KUKA KRL program: MyProgram_189().src

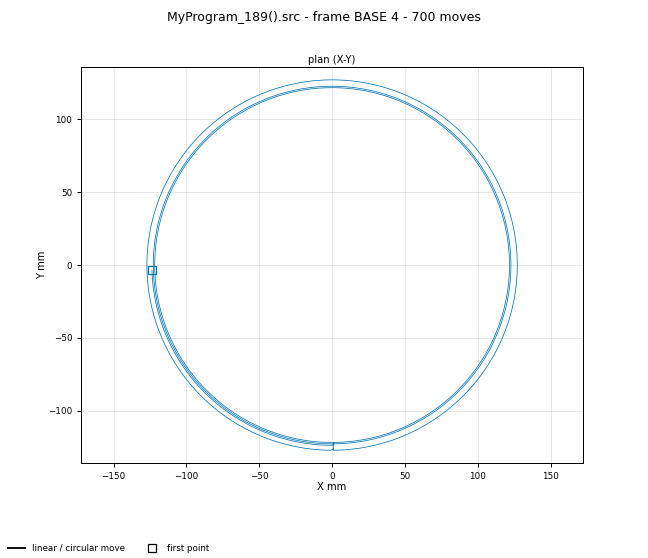
[picture p0: tool path of MyProgram_189().src in frame BASE 4, 700 of 700 moves have a stored position in this frame; points joined in program order, loops and branches not executed]
&ACCESS RVP
&REL 1
&PARAM TEMPLATE = C:\KRC\Roboter\Template\vorgabe
&PARAM EDITMASK = *
DEF MyProgram_189()
; ---- Setting reference (Base) ----
$BASE = BASE_DATA[4]

; --------------------------
; ---- Setting tool (TCP) ----
$TOOL = TOOL_DATA[3]
; --------------------------

$VEL.CP = VEL_APROX_PRINT
Startdeposition()
$VEL.CP = VEL_PRINT
LIN {X -123.6871,Y -3.6269,Z 137,A 178.2903,B 24.9532,C -1.5798,E1 24.8398,E2 627.9376} C_DIS
LIN {X -123.3118,Y -10.2868,Z 137,A -177.6765,B 24.9513,C -1.6119,E1 24.8407,E2 623.8034} C_DIS
LIN {X -122.6788,Y -16.1715,Z 137,A -175.7764,B 24.9541,C -1.5654,E1 24.8413,E2 622.0029} C_DIS
LIN {X -121.5631,Y -23.1085,Z 137,A -172.7109,B 24.9552,C -1.5466,E1 24.8427,E2 618.9641} C_DIS
LIN {X -120.6893,Y -27.3078,Z 137,A -170.7718,B 24.9557,C -1.5382,E1 24.8439,E2 617.0335} C_DIS
LIN {X -120.022,Y -30.1061,Z 137,A -169.137,B 24.9551,C -1.5475,E1 24.8449,E2 615.367} C_DIS
LIN {X -119.1579,Y -33.3607,Z 137,A -167.6264,B 24.9555,C -1.5405,E1 24.8461,E2 613.8643} C_DIS
LIN {X -118.1442,Y -36.7947,Z 137,A -165.8598,B 24.9555,C -1.5402,E1 24.8475,E2 612.0882} C_DIS
LIN {X -116.8715,Y -40.6521,Z 137,A -164.0681,B 24.9561,C -1.5305,E1 24.8491,E2 610.3094} C_DIS
LIN {X -115.0667,Y -45.5133,Z 137,A -161.702,B 24.9566,C -1.5218,E1 24.8514,E2 607.9509} C_DIS
LIN {X -113.3795,Y -49.5667,Z 137,A -159.0001,B 24.9552,C -1.5459,E1 24.8545,E2 605.1764} C_DIS
LIN {X -111.5077,Y -53.6436,Z 137,A -157.538,B 24.9572,C -1.5122,E1 24.8562,E2 603.7867} C_DIS
LIN {X -110.1039,Y -56.4691,Z 137,A -155.9162,B 24.957,C -1.5153,E1 24.8582,E2 602.1488} C_DIS
LIN {X -107.9699,Y -60.4525,Z 137,A -153.8399,B 24.9574,C -1.5088,E1 24.861,E2 600.0772} C_DIS
LIN {X -105.7639,Y -64.2339,Z 137,A -151.6138,B 24.9572,C -1.5123,E1 24.8642,E2 597.8311} C_DIS
LIN {X -103.0515,Y -68.5012,Z 137,A -149.4533,B 24.958,C -1.4979,E1 24.8675,E2 595.694} C_DIS
LIN {X -101.0702,Y -71.3917,Z 137,A -147.7939,B 24.9581,C -1.4955,E1 24.8701,E2 594.0324} C_DIS
LIN {X -98.5873,Y -74.7836,Z 137,A -145.5061,B 24.9575,C -1.5062,E1 24.874,E2 591.708} C_DIS
LIN {X -96.2651,Y -77.7495,Z 137,A -144.2835,B 24.9591,C -1.4782,E1 24.8761,E2 590.5464} C_DIS
LIN {X -94.0528,Y -80.4124,Z 137,A -142.028,B 24.9576,C -1.5042,E1 24.8803,E2 588.2186} C_DIS
LIN {X -91.1944,Y -83.6394,Z 137,A -140.5066,B 24.9591,C -1.4779,E1 24.883,E2 586.7531} C_DIS
LIN {X -88.2872,Y -86.7026,Z 137,A -138.5112,B 24.9592,C -1.4754,E1 24.8869,E2 584.7551} C_DIS
LIN {X -84.7954,Y -90.1202,Z 137,A -136.2459,B 24.9595,C -1.4708,E1 24.8915,E2 582.4914} C_DIS
LIN {X -81.9301,Y -92.733,Z 137,A -134.2054,B 24.9591,C -1.4784,E1 24.8958,E2 580.4245} C_DIS
LIN {X -79.4553,Y -94.8621,Z 137,A -132.7772,B 24.9594,C -1.4716,E1 24.8988,E2 579.007} C_DIS
LIN {X -76.1,Y -97.575,Z 137,A -130.9012,B 24.9599,C -1.4623,E1 24.9029,E2 577.1463} C_DIS
LIN {X -71.8228,Y -100.7645,Z 137,A -128.2909,B 24.9599,C -1.4644,E1 24.9088,E2 574.5216} C_DIS
LIN {X -68.6261,Y -102.9681,Z 137,A -126.6407,B 24.9604,C -1.4546,E1 24.9126,E2 572.8893} C_DIS
LIN {X -63.7724,Y -106.043,Z 137,A -124.2535,B 24.9613,C -1.4378,E1 24.9182,E2 570.5346} C_DIS
LIN {X -60.1181,Y -108.1564,Z 137,A -122.1093,B 24.9609,C -1.4438,E1 24.9234,E2 568.3698} C_DIS
LIN {X -56.5383,Y -110.0687,Z 137,A -120.1188,B 24.9609,C -1.4465,E1 24.9283,E2 566.3673} C_DIS
LIN {X -53.3181,Y -111.6632,Z 137,A -118.5447,B 24.9611,C -1.4403,E1 24.9323,E2 564.8039} C_DIS
LIN {X -50.4843,Y -112.9727,Z 137,A -117.1034,B 24.9612,C -1.4385,E1 24.9359,E2 563.3635} C_DIS
LIN {X -47.5297,Y -114.2474,Z 137,A -115.6287,B 24.9614,C -1.4361,E1 24.9397,E2 561.8909} C_DIS
LIN {X -44.917,Y -115.2996,Z 137,A -114.3059,B 24.9614,C -1.4357,E1 24.9432,E2 560.5662} C_DIS
LIN {X -41.6351,Y -116.5254,Z 137,A -112.6718,B 24.9614,C -1.4348,E1 24.9474,E2 558.931} C_DIS
LIN {X -38.2424,Y -117.6836,Z 137,A -110.1543,B 24.9593,C -1.4744,E1 24.9544,E2 556.3149} C_DIS
LIN {X -32.6953,Y -119.344,Z 137,A -107.5652,B 24.9596,C -1.4682,E1 24.9613,E2 553.7364} C_DIS
LIN {X -27.6129,Y -120.6196,Z 137,A -106.2171,B 24.9625,C -1.4153,E1 24.9647,E2 552.5121} C_DIS
LIN {X -24.7432,Y -121.2408,Z 137,A -104.5438,B 24.9617,C -1.4296,E1 24.9693,E2 550.8029} C_DIS
LIN {X -21.8539,Y -121.7948,Z 137,A -103.1642,B 24.9617,C -1.4299,E1 24.9731,E2 549.421} C_DIS
LIN {X -18.5585,Y -122.3409,Z 137,A -101.5093,B 24.9614,C -1.4347,E1 24.9777,E2 547.7533} C_DIS
LIN {X -14.6586,Y -122.8687,Z 137,A -99.7775,B 24.9617,C -1.43,E1 24.9825,E2 546.0315} C_DIS
LIN {X -10.8263,Y -123.2662,Z 137,A -97.9502,B 24.9616,C -1.4319,E1 24.9876,E2 544.1986} C_DIS
LIN {X -7.19,Y -123.5317,Z 137,A -96.2218,B 24.9615,C -1.4339,E1 24.9924,E2 542.4649} C_DIS
LIN {X -3.2774,Y -123.6968,Z 137,A -94.53,B 24.9618,C -1.4282,E1 24.9971,E2 540.7862} C_DIS
LIN {X 0.3681,Y -123.74,Z 137,A -92.7859,B 24.9616,C -1.4313,E1 25.002,E2 539.0349} C_DIS
LIN {X 0.3681,Y -123.74,Z 137,A -92.7859,B 24.9616,C -1.4313,E1 25.002,E2 539.0349} C_DIS
Enddeposition()
LIN {X 0.8758,Y -122.7486,Z 137,A -93.1134,B 24.7966,C -1.3866,E1 24.8338,E2 539.4449} C_DIS
Startdeposition()
$VEL.CP = VEL_PRINT
LIN {X -2.203,Y -122.7353,Z 137,A -94.7816,B 24.7972,C -1.3754,E1 24.829,E2 541.1399} C_DIS
LIN {X -6.2,Y -122.5983,Z 137,A -96.5836,B 24.797,C -1.3783,E1 24.824,E2 542.9354} C_DIS
LIN {X -10.1585,Y -122.3339,Z 137,A -98.4379,B 24.797,C -1.3782,E1 24.8188,E2 544.7908} C_DIS
LIN {X -13.8748,Y -121.97,Z 137,A -100.0956,B 24.7968,C -1.3823,E1 24.8143,E2 546.4395} C_DIS
LIN {X -16.3768,Y -121.6582,Z 137,A -101.2545,B 24.7968,C -1.3834,E1 24.8111,E2 547.5966} C_DIS
LIN {X -19.0663,Y -121.2654,Z 137,A -102.6876,B 24.7972,C -1.3761,E1 24.8071,E2 549.0485} C_DIS
LIN {X -23.0341,Y -120.5743,Z 137,A -104.5963,B 24.7972,C -1.3755,E1 24.8018,E2 550.9607} C_DIS
LIN {X -26.3906,Y -119.8854,Z 137,A -106.3525,B 24.7975,C -1.3689,E1 24.797,E2 552.7346} C_DIS
LIN {X -31.0253,Y -118.7709,Z 137,A -108.4556,B 24.7972,C -1.3758,E1 24.7913,E2 554.8243} C_DIS
LIN {X -36.1084,Y -117.3239,Z 137,A -110.7655,B 24.7967,C -1.3848,E1 24.7852,E2 557.1166} C_DIS
LIN {X -39.4539,Y -116.2436,Z 137,A -112.57,B 24.797,C -1.3786,E1 24.7803,E2 558.9394} C_DIS
LIN {X -43.2692,Y -114.876,Z 137,A -114.3597,B 24.7967,C -1.385,E1 24.7757,E2 560.7174} C_DIS
LIN {X -47.3278,Y -113.264,Z 137,A -116.3718,B 24.7965,C -1.3883,E1 24.7705,E2 562.7262} C_DIS
LIN {X -50.4824,Y -111.8943,Z 137,A -118.082,B 24.7967,C -1.3853,E1 24.7661,E2 564.4477} C_DIS
LIN {X -54.3057,Y -110.0888,Z 137,A -120.0413,B 24.7965,C -1.3883,E1 24.7611,E2 566.4047} C_DIS
LIN {X -58.3909,Y -107.9802,Z 137,A -122.2379,B 24.7965,C -1.3889,E1 24.7557,E2 568.6062} C_DIS
LIN {X -61.4605,Y -106.2625,Z 137,A -123.6618,B 24.7959,C -1.401,E1 24.7523,E2 570.0052} C_DIS
LIN {X -64.4498,Y -104.4767,Z 137,A -125.4217,B 24.796,C -1.3974,E1 24.7481,E2 571.7793} C_DIS
LIN {X -66.9121,Y -102.9168,Z 137,A -126.6891,B 24.7957,C -1.4037,E1 24.7451,E2 573.0356} C_DIS
LIN {X -70.0256,Y -100.8242,Z 137,A -128.5719,B 24.7959,C -1.4007,E1 24.7408,E2 574.932} C_DIS
LIN {X -73.4065,Y -98.3901,Z 137,A -130.4788,B 24.7956,C -1.4058,E1 24.7365,E2 576.8335} C_DIS
LIN {X -76.3345,Y -96.1362,Z 137,A -132.99,B 24.7973,C -1.3741,E1 24.7308,E2 579.43} C_DIS
LIN {X -80.5143,Y -92.664,Z 137,A -134.5604,B 24.7947,C -1.4218,E1 24.7277,E2 580.8922} C_DIS
LIN {X -82.724,Y -90.6969,Z 137,A -136.647,B 24.7963,C -1.3933,E1 24.7232,E2 583.0555} C_DIS
LIN {X -85.7181,Y -87.8727,Z 137,A -138.0889,B 24.7949,C -1.4185,E1 24.7204,E2 584.4431} C_DIS
LIN {X -88.4014,Y -85.1726,Z 137,A -139.9578,B 24.7949,C -1.4183,E1 24.7167,E2 586.3205} C_DIS
LIN {X -92.3318,Y -80.895,Z 137,A -142.3613,B 24.7939,C -1.4381,E1 24.7123,E2 588.6874} C_DIS
LIN {X -95.0176,Y -77.7224,Z 137,A -144.8359,B 24.7949,C -1.4192,E1 24.7078,E2 591.2188} C_DIS
LIN {X -98.2431,Y -73.6039,Z 137,A -147.0598,B 24.794,C -1.4347,E1 24.704,E2 593.4162} C_DIS
LIN {X -100.2392,Y -70.8606,Z 137,A -148.6789,B 24.794,C -1.4372,E1 24.7014,E2 595.0374} C_DIS
LIN {X -102.6767,Y -67.2806,Z 137,A -150.6986,B 24.7936,C -1.4425,E1 24.6983,E2 597.0544} C_DIS
LIN {X -104.7284,Y -64.0399,Z 137,A -152.4277,B 24.7932,C -1.4499,E1 24.6957,E2 598.7747} C_DIS
LIN {X -106.8253,Y -60.4779,Z 137,A -154.4607,B 24.7932,C -1.4507,E1 24.6929,E2 600.8165} C_DIS
LIN {X -108.9144,Y -56.6265,Z 137,A -156.3406,B 24.7925,C -1.4636,E1 24.6904,E2 602.6756} C_DIS
LIN {X -110.111,Y -54.2606,Z 137,A -157.5975,B 24.7923,C -1.4663,E1 24.6889,E2 603.9328} C_DIS
LIN {X -112.469,Y -49.19,Z 137,A -160.1364,B 24.7917,C -1.4768,E1 24.6859,E2 606.4604} C_DIS
LIN {X -114.1297,Y -45.2066,Z 137,A -162.5726,B 24.7924,C -1.4645,E1 24.6833,E2 608.9399} C_DIS
LIN {X -115.6223,Y -41.2351,Z 137,A -164.2347,B 24.7913,C -1.4842,E1 24.6818,E2 610.5642} C_DIS
LIN {X -116.4754,Y -38.7577,Z 137,A -165.5381,B 24.7913,C -1.4844,E1 24.6806,E2 611.8745} C_DIS
LIN {X -117.6988,Y -34.8687,Z 137,A -167.4771,B 24.7911,C -1.4887,E1 24.679,E2 613.8145} C_DIS
LIN {X -118.6317,Y -31.5472,Z 137,A -169.0788,B 24.7908,C -1.4941,E1 24.6778,E2 615.4128} C_DIS
LIN {X -119.3871,Y -28.5564,Z 137,A -170.4849,B 24.7904,C -1.5,E1 24.6769,E2 616.8129} C_DIS
LIN {X -120.248,Y -24.6815,Z 137,A -172.3898,B 24.7902,C -1.5036,E1 24.6758,E2 618.7204} C_DIS
LIN {X -121.2683,Y -19.0474,Z 137,A -174.8254,B 24.7892,C -1.5223,E1 24.6746,E2 621.1257} C_DIS
LIN {X -121.6872,Y -16.1555,Z 137,A -177.037,B 24.791,C -1.4904,E1 24.6737,E2 623.4272} C_DIS
LIN {X -122.1963,Y -11.6968,Z 137,A -178.4788,B 24.789,C -1.525,E1 24.6734,E2 624.7946} C_DIS
LIN {X -122.6145,Y -5.8764,Z 137,A 178.5874,B 24.789,C -1.5248,E1 24.6728,E2 627.7467} C_DIS
LIN {X -122.7397,Y 1.9378,Z 137,A 174.6848,B 24.789,C -1.5259,E1 24.6728,E2 631.6704} C_DIS
LIN {X -122.64,Y 5.3393,Z 137,A 173.499,B 24.7876,C -1.5483,E1 24.6728,E2 632.8097} C_DIS
LIN {X -122.4564,Y 8.564,Z 137,A 171.4913,B 24.7886,C -1.5319,E1 24.6733,E2 634.8689} C_DIS
LIN {X -122.1415,Y 12.268,Z 137,A 170.293,B 24.7869,C -1.5605,E1 24.6736,E2 636.0059} C_DIS
LIN {X -121.5349,Y 17.2629,Z 137,A 168.0484,B 24.7862,C -1.5726,E1 24.6743,E2 638.2348} C_DIS
LIN {X -121.1308,Y 19.9036,Z 137,A 166.5383,B 24.7866,C -1.5654,E1 24.675,E2 639.7714} C_DIS
LIN {X -120.4521,Y 23.672,Z 137,A 164.4795,B 24.787,C -1.5596,E1 24.6761,E2 641.8564} C_DIS
LIN {X -119.5012,Y 28.0833,Z 137,A 162.5098,B 24.7862,C -1.5722,E1 24.6773,E2 643.8075} C_DIS
LIN {X -118.5997,Y 31.6672,Z 137,A 160.9056,B 24.7856,C -1.583,E1 24.6784,E2 645.3953} C_DIS
LIN {X -117.6401,Y 35.0693,Z 137,A 158.6514,B 24.7868,C -1.5625,E1 24.6802,E2 647.7118} C_DIS
LIN {X -116.3206,Y 39.2222,Z 137,A 157.2285,B 24.7849,C -1.5949,E1 24.6814,E2 649.0649} C_DIS
LIN {X -115.2329,Y 42.3153,Z 137,A 155.3591,B 24.7855,C -1.5852,E1 24.6832,E2 650.9683} C_DIS
LIN {X -113.6971,Y 46.2798,Z 137,A 153.5156,B 24.7847,C -1.5974,E1 24.6851,E2 652.7929} C_DIS
LIN {X -112.1953,Y 49.8095,Z 137,A 151.7129,B 24.7844,C -1.6024,E1 24.6871,E2 654.5937} C_DIS
LIN {X -110.2535,Y 53.9717,Z 137,A 149.805,B 24.7834,C -1.6191,E1 24.6894,E2 656.4721} C_DIS
LIN {X -108.7234,Y 56.9901,Z 137,A 148.0972,B 24.7834,C -1.6183,E1 24.6916,E2 658.1909} C_DIS
LIN {X -104.3676,Y 64.6266,Z 137,A 144.018,B 24.7827,C -1.6313,E1 24.6973,E2 662.2604} C_DIS
LIN {X -100.8109,Y 70.0449,Z 137,A 141.0126,B 24.7821,C -1.6407,E1 24.7019,E2 665.2584} C_DIS
LIN {X -99.122,Y 72.4157,Z 137,A 139.4708,B 24.7823,C -1.6365,E1 24.7044,E2 666.8178} C_DIS
LIN {X -96.7658,Y 75.5356,Z 137,A 137.5795,B 24.7823,C -1.6386,E1 24.7077,E2 668.7132} C_DIS
LIN {X -93.9199,Y 79.0455,Z 137,A 135.5122,B 24.7817,C -1.646,E1 24.7113,E2 670.7723} C_DIS
LIN {X -91.1205,Y 82.2572,Z 137,A 133.4751,B 24.7816,C -1.649,E1 24.7151,E2 672.8114} C_DIS
LIN {X -88.1698,Y 85.4119,Z 137,A 131.4886,B 24.7812,C -1.6554,E1 24.7189,E2 674.7914} C_DIS
LIN {X -85.0909,Y 88.4804,Z 137,A 129.3979,B 24.781,C -1.6576,E1 24.7231,E2 676.8856} C_DIS
LIN {X -81.9678,Y 91.3804,Z 137,A 127.4245,B 24.7807,C -1.663,E1 24.7271,E2 678.8541} C_DIS
LIN {X -78.6966,Y 94.2126,Z 137,A 125.4011,B 24.7804,C -1.6674,E1 24.7314,E2 680.8749} C_DIS
LIN {X -75.4137,Y 96.8605,Z 137,A 123.4335,B 24.7801,C -1.6717,E1 24.7357,E2 682.8394} C_DIS
LIN {X -72.15,Y 99.3151,Z 137,A 121.621,B 24.7796,C -1.6799,E1 24.7398,E2 684.6389} C_DIS
LIN {X -69.1197,Y 101.448,Z 137,A 119.8947,B 24.7794,C -1.6835,E1 24.7437,E2 686.3624} C_DIS
LIN {X -65.9902,Y 103.5106,Z 137,A 117.7864,B 24.7802,C -1.6711,E1 24.7488,E2 688.5072} C_DIS
LIN {X -63.2429,Y 105.2119,Z 137,A 116.8047,B 24.7785,C -1.6971,E1 24.751,E2 689.4298} C_DIS
LIN {X -59.2633,Y 107.5036,Z 137,A 114.3529,B 24.7791,C -1.6873,E1 24.757,E2 691.9123} C_DIS
LIN {X -55.8278,Y 109.3249,Z 137,A 112.1278,B 24.7801,C -1.6723,E1 24.7626,E2 694.1794} C_DIS
LIN {X -52.1225,Y 111.1411,Z 137,A 110.6447,B 24.7787,C -1.6949,E1 24.7662,E2 695.6123} C_DIS
LIN {X -48.0117,Y 112.9784,Z 137,A 108.6136,B 24.7783,C -1.7012,E1 24.7714,E2 697.6333} C_DIS
LIN {X -45.7892,Y 113.8948,Z 137,A 107.4863,B 24.7782,C -1.7025,E1 24.7743,E2 698.7598} C_DIS
LIN {X -42.6178,Y 115.12,Z 137,A 105.6898,B 24.7786,C -1.6953,E1 24.7791,E2 700.5774} C_DIS
LIN {X -38.9692,Y 116.405,Z 137,A 104.0227,B 24.7781,C -1.7037,E1 24.7834,E2 702.2275} C_DIS
LIN {X -35.2511,Y 117.5863,Z 137,A 102.2728,B 24.7777,C -1.709,E1 24.7881,E2 703.9679} C_DIS
LIN {X -32.0652,Y 118.4936,Z 137,A 100.5251,B 24.7782,C -1.7016,E1 24.7928,E2 705.7361} C_DIS
LIN {X -25.034,Y 120.1753,Z 137,A 97.1526,B 24.778,C -1.7048,E1 24.802,E2 709.1054} C_DIS
LIN {X -20.6937,Y 120.999,Z 137,A 95.0483,B 24.778,C -1.7045,E1 24.8078,E2 711.2126} C_DIS
LIN {X -15.9129,Y 121.719,Z 137,A 92.9545,B 24.7775,C -1.7133,E1 24.8135,E2 713.2869} C_DIS
LIN {X -11.9129,Y 122.1756,Z 137,A 91.0049,B 24.7776,C -1.7111,E1 24.8189,E2 715.2429} C_DIS
LIN {X -8.3225,Y 122.474,Z 137,A 89.2904,B 24.7776,C -1.7103,E1 24.8237,E2 716.96} C_DIS
LIN {X -4.1345,Y 122.687,Z 137,A 87.3465,B 24.7776,C -1.7116,E1 24.8291,E2 718.9014} C_DIS
LIN {X 0.1125,Y 122.7562,Z 137,A 85.5481,B 24.777,C -1.7205,E1 24.8341,E2 720.6785} C_DIS
LIN {X 2.9118,Y 122.7214,Z 137,A 84.0821,B 24.7775,C -1.7133,E1 24.8382,E2 722.1613} C_DIS
LIN {X 6.6577,Y 122.5752,Z 137,A 82.257,B 24.7777,C -1.7099,E1 24.8434,E2 723.9939} C_DIS
LIN {X 10.6566,Y 122.2919,Z 137,A 80.5997,B 24.7771,C -1.7197,E1 24.8479,E2 725.6272} C_DIS
LIN {X 13.2057,Y 122.0425,Z 137,A 79.41,B 24.7771,C -1.7198,E1 24.8512,E2 726.8158} C_DIS
LIN {X 16.416,Y 121.6531,Z 137,A 77.7186,B 24.7776,C -1.711,E1 24.8559,E2 728.5268} C_DIS
LIN {X 22.1969,Y 120.7326,Z 137,A 75.2128,B 24.777,C -1.7206,E1 24.8628,E2 731.0073} C_DIS
LIN {X 25.0485,Y 120.1732,Z 137,A 73.8008,B 24.7772,C -1.7174,E1 24.8667,E2 732.4251} C_DIS
LIN {X 28.6066,Y 119.375,Z 137,A 72.0632,B 24.7774,C -1.7148,E1 24.8714,E2 734.1665} C_DIS
LIN {X 32.9824,Y 118.2407,Z 137,A 69.932,B 24.7775,C -1.7124,E1 24.8772,E2 736.3} C_DIS
LIN {X 36.4139,Y 117.2305,Z 137,A 68.1877,B 24.7778,C -1.7076,E1 24.8818,E2 738.0525} C_DIS
LIN {X 40.391,Y 115.9193,Z 137,A 66.3001,B 24.7778,C -1.7091,E1 24.8868,E2 739.9329} C_DIS
LIN {X 43.2459,Y 114.8847,Z 137,A 64.9095,B 24.7778,C -1.7091,E1 24.8904,E2 741.3207} C_DIS
LIN {X 46.9033,Y 113.4413,Z 137,A 63.0239,B 24.778,C -1.7047,E1 24.8953,E2 743.2124} C_DIS
LIN {X 50.1295,Y 112.0522,Z 137,A 61.4129,B 24.778,C -1.7042,E1 24.8995,E2 744.8206} C_DIS
LIN {X 53.7956,Y 110.3404,Z 137,A 59.6711,B 24.7778,C -1.7089,E1 24.9038,E2 746.5468} C_DIS
LIN {X 55.788,Y 109.3451,Z 137,A 58.4536,B 24.7784,C -1.6991,E1 24.9069,E2 747.7843} C_DIS
LIN {X 58.6867,Y 107.8193,Z 137,A 56.9474,B 24.7784,C -1.698,E1 24.9106,E2 749.2886} C_DIS
LIN {X 62.5269,Y 105.6391,Z 137,A 54.9522,B 24.7784,C -1.6981,E1 24.9154,E2 751.2775} C_DIS
LIN {X 65.6556,Y 103.7231,Z 137,A 52.9293,B 24.7796,C -1.6806,E1 24.9203,E2 753.3355} C_DIS
LIN {X 70.0314,Y 100.8202,Z 137,A 50.8892,B 24.7786,C -1.6962,E1 24.9249,E2 755.3316} C_DIS
LIN {X 72.9166,Y 98.754,Z 137,A 49.0242,B 24.7794,C -1.6832,E1 24.9292,E2 757.2208} C_DIS
LIN {X 77.6234,Y 95.0985,Z 137,A 46.3169,B 24.7795,C -1.6816,E1 24.9351,E2 759.9218} C_DIS
LIN {X 80.7677,Y 92.4429,Z 137,A 44.3862,B 24.7798,C -1.6773,E1 24.9392,E2 761.8551} C_DIS
LIN {X 83.9408,Y 89.5723,Z 137,A 42.3367,B 24.7802,C -1.6707,E1 24.9434,E2 763.9121} C_DIS
LIN {X 87.1045,Y 86.498,Z 137,A 40.3419,B 24.7802,C -1.6693,E1 24.9474,E2 765.9016} C_DIS
LIN {X 91.2923,Y 82.0662,Z 137,A 37.6862,B 24.7802,C -1.6722,E1 24.9524,E2 768.5389} C_DIS
LIN {X 93.0147,Y 80.1085,Z 137,A 36.2748,B 24.7809,C -1.6598,E1 24.955,E2 769.9731} C_DIS
LIN {X 95.8384,Y 76.7086,Z 137,A 34.2601,B 24.781,C -1.6572,E1 24.9586,E2 771.9847} C_DIS
LIN {X 98.3214,Y 73.4987,Z 137,A 32.1112,B 24.7821,C -1.6401,E1 24.9622,E2 774.1639} C_DIS
LIN {X 100.2318,Y 70.8711,Z 137,A 31.0152,B 24.7811,C -1.6568,E1 24.9639,E2 775.2149} C_DIS
LIN {X 102.3733,Y 67.7414,Z 137,A 29.0594,B 24.7819,C -1.643,E1 24.967,E2 777.1936} C_DIS
LIN {X 104.827,Y 63.8792,Z 137,A 26.9377,B 24.7822,C -1.638,E1 24.9702,E2 779.3163} C_DIS
LIN {X 107.0081,Y 60.153,Z 137,A 25.1524,B 24.7819,C -1.6438,E1 24.9726,E2 781.0785} C_DIS
LIN {X 108.1589,Y 58.0583,Z 137,A 23.817,B 24.7827,C -1.6299,E1 24.9744,E2 782.44} C_DIS
LIN {X 109.6734,Y 55.1431,Z 137,A 22.4667,B 24.7825,C -1.6346,E1 24.9761,E2 783.7719} C_DIS
LIN {X 111.0312,Y 52.3555,Z 137,A 20.789,B 24.7834,C -1.619,E1 24.9782,E2 785.4774} C_DIS
LIN {X 112.6018,Y 48.8828,Z 137,A 19.2077,B 24.7831,C -1.6236,E1 24.9799,E2 787.0391} C_DIS
LIN {X 113.9256,Y 45.7128,Z 137,A 17.5903,B 24.7835,C -1.6182,E1 24.9817,E2 788.6604} C_DIS
LIN {X 115.0761,Y 42.735,Z 137,A 16.0482,B 24.7839,C -1.6112,E1 24.9832,E2 790.2106} C_DIS
LIN {X 116.3876,Y 39.0214,Z 137,A 13.7827,B 24.7855,C -1.5845,E1 24.9853,E2 792.5264} C_DIS
LIN {X 117.6652,Y 34.9834,Z 137,A 12.4794,B 24.7839,C -1.6117,E1 24.9863,E2 793.7576} C_DIS
LIN {X 118.7237,Y 31.2024,Z 137,A 10.5437,B 24.7845,C -1.6009,E1 24.9877,E2 795.7078} C_DIS
LIN {X 119.8092,Y 26.7336,Z 137,A 8.3035,B 24.7852,C -1.5895,E1 24.9892,E2 797.962} C_DIS
LIN {X 120.6603,Y 22.5841,Z 137,A 6.4845,B 24.7852,C -1.5911,E1 24.9901,E2 799.7665} C_DIS
LIN {X 121.2382,Y 19.2418,Z 137,A 4.7936,B 24.7857,C -1.5807,E1 24.9909,E2 801.4721} C_DIS
LIN {X 121.7539,Y 15.6468,Z 137,A 3.0442,B 24.7862,C -1.5725,E1 24.9916,E2 803.2305} C_DIS
LIN {X 122.1977,Y 11.6825,Z 137,A 1.3084,B 24.7862,C -1.5728,E1 24.9921,E2 804.9553} C_DIS
LIN {X 122.4698,Y 8.3798,Z 137,A -0.3302,B 24.7868,C -1.5631,E1 24.9924,E2 806.607} C_DIS
LIN {X 122.6717,Y 4.526,Z 137,A -2.1209,B 24.7871,C -1.5578,E1 24.9926,E2 808.3997} C_DIS
LIN {X 122.7585,Y 0,Z 137,A -4.3029,B 24.7877,C -1.5473,E1 24.9926,E2 810.5933} C_DIS
LIN {X 122.7047,Y -3.5131,Z 137,A -5.8087,B 24.7877,C -1.5487,E1 24.9926,E2 812.0869} C_DIS
LIN {X 122.5222,Y -7.5547,Z 137,A -7.6258,B 24.7877,C -1.5461,E1 24.9923,E2 813.8993} C_DIS
LIN {X 122.291,Y -10.6673,Z 137,A -9.1396,B 24.7882,C -1.5384,E1 24.992,E2 815.4222} C_DIS
LIN {X 121.8916,Y -14.5318,Z 137,A -10.9458,B 24.7885,C -1.5329,E1 24.9914,E2 817.2309} C_DIS
LIN {X 121.3522,Y -18.5057,Z 137,A -12.7501,B 24.7887,C -1.5301,E1 24.9907,E2 819.0309} C_DIS
LIN {X 120.7435,Y -22.1362,Z 137,A -14.731,B 24.7898,C -1.5113,E1 24.9897,E2 821.0447} C_DIS
LIN {X 120.123,Y -25.2897,Z 137,A -15.8209,B 24.7889,C -1.527,E1 24.9891,E2 822.0911} C_DIS
LIN {X 119.1663,Y -29.4724,Z 137,A -17.8529,B 24.7893,C -1.519,E1 24.9878,E2 824.1302} C_DIS
LIN {X 118.415,Y -32.359,Z 137,A -19.4853,B 24.7903,C -1.5025,E1 24.9866,E2 825.7923} C_DIS
LIN {X 116.9519,Y -37.2953,Z 137,A -21.4782,B 24.7896,C -1.5154,E1 24.985,E2 827.7431} C_DIS
LIN {X 116.2366,Y -39.4747,Z 137,A -22.8911,B 24.7907,C -1.4948,E1 24.9837,E2 829.1968} C_DIS
LIN {X 115.0726,Y -42.7444,Z 137,A -24.4034,B 24.7907,C -1.4951,E1 24.9823,E2 830.7} C_DIS
LIN {X 113.7474,Y -46.1549,Z 137,A -26.0034,B 24.7907,C -1.4951,E1 24.9807,E2 832.2909} C_DIS
LIN {X 110.5136,Y -53.439,Z 137,A -29.6528,B 24.7912,C -1.4871,E1 24.9765,E2 835.9392} C_DIS
LIN {X 109.3774,Y -55.7246,Z 137,A -31.5393,B 24.7933,C -1.449,E1 24.974,E2 837.9062} C_DIS
LIN {X 107.1276,Y -59.9403,Z 137,A -33.0542,B 24.7917,C -1.4778,E1 24.9721,E2 839.3447} C_DIS
LIN {X 105.3215,Y -63.0599,Z 137,A -34.8601,B 24.7923,C -1.4667,E1 24.9695,E2 841.1676} C_DIS
LIN {X 103.1482,Y -66.5558,Z 137,A -36.824,B 24.7927,C -1.459,E1 24.9665,E2 843.1397} C_DIS
LIN {X 100.7451,Y -70.1394,Z 137,A -38.8034,B 24.7929,C -1.455,E1 24.9634,E2 845.1188} C_DIS
LIN {X 98.4075,Y -73.3831,Z 137,A -40.6198,B 24.7931,C -1.4523,E1 24.9604,E2 846.9328} C_DIS
LIN {X 95.2985,Y -77.3786,Z 137,A -42.8045,B 24.793,C -1.4547,E1 24.9567,E2 849.1014} C_DIS
LIN {X 93.2528,Y -79.832,Z 137,A -44.5306,B 24.7938,C -1.4391,E1 24.9535,E2 850.8566} C_DIS
LIN {X 90.2798,Y -83.1786,Z 137,A -46.6082,B 24.7941,C -1.4343,E1 24.9496,E2 852.9363} C_DIS
LIN {X 87.4909,Y -86.1074,Z 137,A -48.424,B 24.7941,C -1.4331,E1 24.9461,E2 854.7472} C_DIS
LIN {X 84.8779,Y -88.684,Z 137,A -50.0681,B 24.7941,C -1.4323,E1 24.9428,E2 856.3862} C_DIS
LIN {X 82.0727,Y -91.2865,Z 137,A -51.8826,B 24.7945,C -1.4266,E1 24.9391,E2 858.2068} C_DIS
LIN {X 78.3435,Y -94.5061,Z 137,A -54.0439,B 24.7945,C -1.4282,E1 24.9345,E2 860.356} C_DIS
LIN {X 75.4968,Y -96.796,Z 137,A -55.9183,B 24.7951,C -1.416,E1 24.9303,E2 862.2521} C_DIS
LIN {X 72.2407,Y -99.2494,Z 137,A -57.8069,B 24.7952,C -1.4127,E1 24.9261,E2 864.1419} C_DIS
LIN {X 69.2251,Y -101.3759,Z 137,A -59.5396,B 24.7954,C -1.4086,E1 24.9221,E2 865.8782} C_DIS
LIN {X 66.4875,Y -103.1923,Z 137,A -61.0685,B 24.7956,C -1.4058,E1 24.9185,E2 867.4088} C_DIS
LIN {X 62.8524,Y -105.4452,Z 137,A -63.2558,B 24.7963,C -1.3927,E1 24.9132,E2 869.6203} C_DIS
LIN {X 56.0614,Y -109.2059,Z 137,A -66.3804,B 24.7953,C -1.4106,E1 24.9057,E2 872.6934} C_DIS
LIN {X 53.8526,Y -110.3123,Z 137,A -68.0298,B 24.7967,C -1.3846,E1 24.9014,E2 874.4001} C_DIS
LIN {X 50.862,Y -111.7239,Z 137,A -69.2093,B 24.7959,C -1.3998,E1 24.8985,E2 875.5406} C_DIS
LIN {X 48.6259,Y -112.7128,Z 137,A -70.4056,B 24.7962,C -1.3954,E1 24.8955,E2 876.7445} C_DIS
LIN {X 45.364,Y -114.0662,Z 137,A -71.9715,B 24.7961,C -1.397,E1 24.8914,E2 878.3029} C_DIS
LIN {X 43.1192,Y -114.9322,Z 137,A -73.1837,B 24.7964,C -1.3911,E1 24.8882,E2 879.5264} C_DIS
LIN {X 39.4137,Y -116.257,Z 137,A -75.5199,B 24.7977,C -1.3648,E1 24.8819,E2 881.9207} C_DIS
LIN {X 35.3682,Y -117.5505,Z 137,A -77.0445,B 24.7967,C -1.3843,E1 24.878,E2 883.396} C_DIS
LIN {X 31.3739,Y -118.6779,Z 137,A -78.8613,B 24.7965,C -1.388,E1 24.8731,E2 885.2011} C_DIS
LIN {X 28.0061,Y -119.5192,Z 137,A -81.1224,B 24.7982,C -1.3559,E1 24.8668,E2 887.5355} C_DIS
LIN {X 23.528,Y -120.4798,Z 137,A -82.4945,B 24.7964,C -1.3904,E1 24.8633,E2 888.8237} C_DIS
LIN {X 20.7444,Y -120.9905,Z 137,A -84.0314,B 24.797,C -1.379,E1 24.8589,E2 890.386} C_DIS
LIN {X 17.1885,Y -121.5456,Z 137,A -85.6821,B 24.797,C -1.3792,E1 24.8544,E2 892.0346} C_DIS
LIN {X 13.1616,Y -122.0472,Z 137,A -87.5274,B 24.797,C -1.3804,E1 24.8493,E2 893.8758} C_DIS
LIN {X 9.1752,Y -122.4117,Z 137,A -89.4488,B 24.7971,C -1.3769,E1 24.8439,E2 895.8044} C_DIS
LIN {X 5.2921,Y -122.6419,Z 137,A -91.2879,B 24.7972,C -1.3751,E1 24.8388,E2 897.6472} C_DIS
LIN {X 1.5361,Y -122.7464,Z 137,A -93.0802,B 24.7973,C -1.3727,E1 24.8338,E2 899.4449} C_DIS
LIN {X 1.5361,Y -122.7464,Z 137,A -93.0802,B 24.7973,C -1.3727,E1 24.8338,E2 899.4449} C_DIS
Enddeposition()
LIN {X 0.8692,Y -121.766,Z 137,A -92.8307,B 24.3643,C -1.3268,E1 24.3996,E2 899.2452} C_DIS
Startdeposition()
$VEL.CP = VEL_PRINT
LIN {X 3.5856,Y -121.7171,Z 137,A -91.0945,B 24.3632,C -1.3484,E1 24.4046,E2 897.457} C_DIS
LIN {X 7.6138,Y -121.5315,Z 137,A -89.323,B 24.3635,C -1.3433,E1 24.4095,E2 895.6984} C_DIS
LIN {X 10.4459,Y -121.321,Z 137,A -87.9539,B 24.3634,C -1.3454,E1 24.4133,E2 894.3248} C_DIS
LIN {X 13.562,Y -121.0132,Z 137,A -86.526,B 24.3634,C -1.3441,E1 24.4173,E2 892.901} C_DIS
LIN {X 16.3802,Y -120.6642,Z 137,A -85.0376,B 24.363,C -1.3521,E1 24.4215,E2 891.3945} C_DIS
LIN {X 19.862,Y -120.1389,Z 137,A -83.7154,B 24.3638,C -1.3377,E1 24.425,E2 890.1087} C_DIS
LIN {X 22.4293,Y -119.6868,Z 137,A -82.1782,B 24.363,C -1.3533,E1 24.4293,E2 888.5355} C_DIS
LIN {X 25.3824,Y -119.0951,Z 137,A -80.9282,B 24.3633,C -1.3466,E1 24.4327,E2 887.3031} C_DIS
LIN {X 28.1451,Y -118.4728,Z 137,A -79.5515,B 24.3631,C -1.35,E1 24.4365,E2 885.9203} C_DIS
LIN {X 31.1747,Y -117.7114,Z 137,A -78.087,B 24.3631,C -1.3513,E1 24.4404,E2 884.4549} C_DIS
LIN {X 34.6069,Y -116.7489,Z 137,A -76.2479,B 24.3626,C -1.3608,E1 24.4454,E2 882.5959} C_DIS
LIN {X 38.1741,Y -115.6314,Z 137,A -74.6151,B 24.3628,C -1.357,E1 24.4497,E2 880.9756} C_DIS
LIN {X 41.017,Y -114.6537,Z 137,A -73.2082,B 24.3627,C -1.3585,E1 24.4534,E2 879.5681} C_DIS
LIN {X 43.959,Y -113.5579,Z 137,A -71.7774,B 24.3627,C -1.3583,E1 24.4572,E2 878.1409} C_DIS
LIN {X 47.1516,Y -112.2699,Z 137,A -70.2578,B 24.3628,C -1.3558,E1 24.4611,E2 876.6307} C_DIS
LIN {X 49.3394,Y -111.3263,Z 137,A -69.0039,B 24.3624,C -1.3639,E1 24.4643,E2 875.3605} C_DIS
LIN {X 52.6353,Y -109.8057,Z 137,A -67.2881,B 24.3622,C -1.367,E1 24.4686,E2 873.6418} C_DIS
LIN {X 56.1918,Y -108.0298,Z 137,A -65.5642,B 24.3624,C -1.3631,E1 24.4729,E2 871.9322} C_DIS
LIN {X 58.6667,Y -106.7078,Z 137,A -64.1352,B 24.362,C -1.3706,E1 24.4764,E2 870.4892} C_DIS
LIN {X 61.2177,Y -105.2646,Z 137,A -62.7422,B 24.3619,C -1.3738,E1 24.4798,E2 869.0929} C_DIS
LIN {X 64.6585,Y -103.1873,Z 137,A -60.7475,B 24.3614,C -1.3824,E1 24.4846,E2 867.0839} C_DIS
LIN {X 68.0307,Y -100.9955,Z 137,A -59.0751,B 24.3618,C -1.3755,E1 24.4884,E2 865.4338} C_DIS
LIN {X 70.239,Y -99.472,Z 137,A -57.7651,B 24.3615,C -1.3804,E1 24.4915,E2 864.1165} C_DIS
LIN {X 72.6551,Y -97.7212,Z 137,A -56.2329,B 24.361,C -1.3896,E1 24.4949,E2 862.5677} C_DIS
LIN {X 76.1408,Y -95.0312,Z 137,A -54.1543,B 24.3608,C -1.3945,E1 24.4995,E2 860.4854} C_DIS
LIN {X 79.542,Y -92.2024,Z 137,A -52.0771,B 24.3605,C -1.399,E1 24.5039,E2 858.4054} C_DIS
LIN {X 82.8755,Y -89.2181,Z 137,A -49.9887,B 24.3603,C -1.4032,E1 24.5083,E2 856.3157} C_DIS
LIN {X 86.0967,Y -86.1145,Z 137,A -47.8823,B 24.36,C -1.4084,E1 24.5125,E2 854.2057} C_DIS
LIN {X 89.2184,Y -82.8752,Z 137,A -45.7825,B 24.3598,C -1.4129,E1 24.5165,E2 852.1044} C_DIS
LIN {X 92.2028,Y -79.5414,Z 137,A -43.6949,B 24.3595,C -1.4175,E1 24.5203,E2 850.0153} C_DIS
LIN {X 95.0622,Y -76.1018,Z 137,A -41.5939,B 24.3592,C -1.423,E1 24.5241,E2 847.9113} C_DIS
LIN {X 97.808,Y -72.5386,Z 137,A -39.6467,B 24.3594,C -1.4204,E1 24.5273,E2 845.9797} C_DIS
LIN {X 99.556,Y -70.1199,Z 137,A -38.2271,B 24.3591,C -1.4251,E1 24.5296,E2 844.5559} C_DIS
LIN {X 101.7262,Y -66.9327,Z 137,A -36.3888,B 24.3588,C -1.4314,E1 24.5325,E2 842.7117} C_DIS
LIN {X 103.6716,Y -63.8784,Z 137,A -34.7243,B 24.3586,C -1.4344,E1 24.535,E2 841.0487} C_DIS
LIN {X 105.206,Y -61.3191,Z 137,A -33.3263,B 24.3584,C -1.4382,E1 24.5369,E2 839.6489} C_DIS
LIN {X 107.0724,Y -57.9986,Z 137,A -31.4172,B 24.3578,C -1.4493,E1 24.5395,E2 837.7233} C_DIS
LIN {X 109.0249,Y -54.2353,Z 137,A -29.7437,B 24.3583,C -1.4395,E1 24.5416,E2 836.0826} C_DIS
LIN {X 110.0735,Y -52.0749,Z 137,A -28.4634,B 24.3577,C -1.4503,E1 24.5432,E2 834.7833} C_DIS
LIN {X 111.3118,Y -49.3719,Z 137,A -27.0221,B 24.3573,C -1.4567,E1 24.5448,E2 833.3347} C_DIS
LIN {X 112.5026,Y -46.5944,Z 137,A -25.6747,B 24.3573,C -1.4574,E1 24.5463,E2 831.9931} C_DIS
LIN {X 113.6103,Y -43.8243,Z 137,A -24.2644,B 24.357,C -1.4621,E1 24.5477,E2 830.5795} C_DIS
LIN {X 114.6532,Y -41.0183,Z 137,A -22.8661,B 24.3568,C -1.466,E1 24.5491,E2 829.1798} C_DIS
LIN {X 115.6698,Y -38.0588,Z 137,A -21.3368,B 24.3564,C -1.4735,E1 24.5504,E2 827.6414} C_DIS
LIN {X 116.5719,Y -35.1993,Z 137,A -20.0344,B 24.3564,C -1.4726,E1 24.5515,E2 826.3487} C_DIS
LIN {X 117.3595,Y -32.4753,Z 137,A -18.6823,B 24.3562,C -1.4778,E1 24.5525,E2 824.9921} C_DIS
LIN {X 118.1551,Y -29.4525,Z 137,A -17.239,B 24.356,C -1.4812,E1 24.5535,E2 823.5493} C_DIS
LIN {X 118.809,Y -26.6913,Z 137,A -15.9139,B 24.3557,C -1.485,E1 24.5544,E2 822.2229} C_DIS
LIN {X 119.4267,Y -23.7767,Z 137,A -14.4549,B 24.3553,C -1.4923,E1 24.5552,E2 820.7548} C_DIS
LIN {X 120.0977,Y -20.1092,Z 137,A -12.9639,B 24.3557,C -1.4851,E1 24.5559,E2 819.2904} C_DIS
LIN {X 120.475,Y -17.7158,Z 137,A -11.6838,B 24.3551,C -1.4957,E1 24.5564,E2 817.9924} C_DIS
LIN {X 120.8552,Y -14.9027,Z 137,A -10.2111,B 24.3545,C -1.5068,E1 24.557,E2 816.5019} C_DIS
LIN {X 121.1976,Y -11.7903,Z 137,A -8.8865,B 24.3546,C -1.5043,E1 24.5573,E2 815.1914} C_DIS
LIN {X 121.4396,Y -8.9605,Z 137,A -7.3732,B 24.3539,C -1.5174,E1 24.5577,E2 813.6557} C_DIS
LIN {X 121.6537,Y -5.3495,Z 137,A -5.8956,B 24.3542,C -1.5118,E1 24.5579,E2 812.2006} C_DIS
LIN {X 121.7379,Y -2.8389,Z 137,A -4.6752,B 24.3539,C -1.5176,E1 24.5579,E2 810.9737} C_DIS
LIN {X 121.7733,Y 0,Z 137,A -3.2549,B 24.3534,C -1.5261,E1 24.558,E2 809.5416} C_DIS
LIN {X 121.7338,Y 2.9844,Z 137,A -1.8291,B 24.353,C -1.5318,E1 24.558,E2 808.1108} C_DIS
LIN {X 121.5752,Y 6.9053,Z 137,A -0.1756,B 24.3532,C -1.5282,E1 24.5577,E2 806.4759} C_DIS
LIN {X 121.3206,Y 10.4496,Z 137,A 1.5458,B 24.3528,C -1.5361,E1 24.5573,E2 804.7461} C_DIS
LIN {X 121.0131,Y 13.5638,Z 137,A 3.0005,B 24.3525,C -1.54,E1 24.5569,E2 803.2909} C_DIS
LIN {X 120.5585,Y 17.1315,Z 137,A 4.7302,B 24.3521,C -1.5473,E1 24.5563,E2 801.5541} C_DIS
LIN {X 120.0027,Y 20.678,Z 137,A 6.4712,B 24.3516,C -1.5552,E1 24.5555,E2 799.8045} C_DIS
LIN {X 119.2965,Y 24.4169,Z 137,A 8.0129,B 24.352,C -1.5486,E1 24.5547,E2 798.2879} C_DIS
LIN {X 118.8201,Y 26.6425,Z 137,A 9.2348,B 24.3514,C -1.5594,E1 24.5539,E2 797.0473} C_DIS
LIN {X 118.12,Y 29.5906,Z 137,A 10.6733,B 24.3511,C -1.5645,E1 24.553,E2 795.6051} C_DIS
LIN {X 117.3214,Y 32.6116,Z 137,A 12.0503,B 24.3511,C -1.5645,E1 24.552,E2 794.2363} C_DIS
LIN {X 116.4883,Y 35.4723,Z 137,A 13.4428,B 24.3508,C -1.5683,E1 24.5508,E2 792.8427} C_DIS
LIN {X 115.4153,Y 38.8228,Z 137,A 15.0469,B 24.3507,C -1.5708,E1 24.5495,E2 791.2419} C_DIS
LIN {X 114.6513,Y 41.0236,Z 137,A 16.2559,B 24.3502,C -1.5796,E1 24.5483,E2 790.0187} C_DIS
LIN {X 113.5589,Y 43.9566,Z 137,A 17.6797,B 24.35,C -1.5816,E1 24.5469,E2 788.5981} C_DIS
LIN {X 112.5031,Y 46.5933,Z 137,A 19.0734,B 24.3496,C -1.5884,E1 24.5454,E2 787.1961} C_DIS
LIN {X 111.1592,Y 49.7131,Z 137,A 20.5329,B 24.3497,C -1.5862,E1 24.5438,E2 785.7499} C_DIS
LIN {X 110.0115,Y 52.2045,Z 137,A 21.8755,B 24.3494,C -1.5925,E1 24.5422,E2 784.3998} C_DIS
LIN {X 108.6997,Y 54.8842,Z 137,A 23.2691,B 24.3492,C -1.5959,E1 24.5405,E2 783.0055} C_DIS
LIN {X 107.392,Y 57.404,Z 137,A 24.5962,B 24.349,C -1.5992,E1 24.5387,E2 781.6776} C_DIS
LIN {X 105.8823,Y 60.143,Z 137,A 26.2084,B 24.3483,C -1.6101,E1 24.5365,E2 780.0478} C_DIS
LIN {X 103.5961,Y 64.0016,Z 137,A 28.1949,B 24.3483,C -1.6097,E1 24.5337,E2 778.0725} C_DIS
LIN {X 101.9926,Y 66.5265,Z 137,A 29.5628,B 24.3482,C -1.6115,E1 24.5316,E2 776.7074} C_DIS
LIN {X 100.3281,Y 69.0108,Z 137,A 30.9624,B 24.348,C -1.6148,E1 24.5294,E2 775.307} C_DIS
LIN {X 98.614,Y 71.4387,Z 137,A 32.4517,B 24.3475,C -1.6228,E1 24.527,E2 773.8059} C_DIS
LIN {X 95.9997,Y 74.916,Z 137,A 34.5517,B 24.347,C -1.6304,E1 24.5234,E2 771.6978} C_DIS
LIN {X 93.1348,Y 78.4484,Z 137,A 36.6649,B 24.3468,C -1.6342,E1 24.5196,E2 769.5854} C_DIS
LIN {X 90.3068,Y 81.6878,Z 137,A 38.6392,B 24.3466,C -1.6365,E1 24.516,E2 767.6146} C_DIS
LIN {X 87.627,Y 84.5561,Z 137,A 40.5008,B 24.3463,C -1.6413,E1 24.5124,E2 765.7497} C_DIS
LIN {X 84.503,Y 87.6785,Z 137,A 42.5995,B 24.346,C -1.6467,E1 24.5082,E2 763.6469} C_DIS
LIN {X 81.2233,Y 90.7247,Z 137,A 44.6904,B 24.3457,C -1.6503,E1 24.5039,E2 761.556} C_DIS
LIN {X 77.8434,Y 93.6411,Z 137,A 46.7779,B 24.3455,C -1.6538,E1 24.4994,E2 759.4685} C_DIS
LIN {X 74.3254,Y 96.4575,Z 137,A 48.9014,B 24.3453,C -1.6579,E1 24.4947,E2 757.3431} C_DIS
LIN {X 71.3345,Y 98.6894,Z 137,A 50.4893,B 24.3456,C -1.653,E1 24.4912,E2 755.7729} C_DIS
LIN {X 68.7046,Y 100.5382,Z 137,A 51.9553,B 24.3456,C -1.6534,E1 24.4879,E2 754.3111} C_DIS
LIN {X 66.2952,Y 102.1428,Z 137,A 53.4865,B 24.3449,C -1.6636,E1 24.4842,E2 752.7604} C_DIS
LIN {X 62.4824,Y 104.5188,Z 137,A 55.5424,B 24.3449,C -1.6641,E1 24.4794,E2 750.7099} C_DIS
LIN {X 59.8888,Y 106.0264,Z 137,A 56.8604,B 24.345,C -1.6617,E1 24.4762,E2 749.4017} C_DIS
LIN {X 57.4021,Y 107.3931,Z 137,A 58.2238,B 24.3448,C -1.6649,E1 24.4728,E2 748.0346} C_DIS
LIN {X 54.7533,Y 108.7664,Z 137,A 59.6023,B 24.3448,C -1.6656,E1 24.4694,E2 746.6585} C_DIS
LIN {X 52.0717,Y 110.075,Z 137,A 61.0124,B 24.3446,C -1.6676,E1 24.4658,E2 745.2472} C_DIS
LIN {X 48.6483,Y 111.6298,Z 137,A 62.8263,B 24.3444,C -1.6717,E1 24.4612,E2 743.4279} C_DIS
LIN {X 46.1241,Y 112.6975,Z 137,A 64.2597,B 24.3439,C -1.6798,E1 24.4575,E2 741.9784} C_DIS
LIN {X 42.2885,Y 114.1913,Z 137,A 65.9951,B 24.3443,C -1.6723,E1 24.453,E2 740.2649} C_DIS
LIN {X 39.4771,Y 115.1934,Z 137,A 67.4981,B 24.344,C -1.6782,E1 24.449,E2 738.7509} C_DIS
LIN {X 35.2158,Y 116.5668,Z 137,A 69.4698,B 24.3443,C -1.6736,E1 24.4438,E2 736.794} C_DIS
LIN {X 32.4867,Y 117.3563,Z 137,A 70.9053,B 24.3439,C -1.6791,E1 24.4399,E2 735.3477} C_DIS
LIN {X 29.4461,Y 118.1567,Z 137,A 72.3199,B 24.344,C -1.677,E1 24.4361,E2 733.9403} C_DIS
LIN {X 26.6871,Y 118.8099,Z 137,A 73.6239,B 24.344,C -1.6763,E1 24.4325,E2 732.6398} C_DIS
LIN {X 23.741,Y 119.434,Z 137,A 75.0419,B 24.344,C -1.677,E1 24.4287,E2 731.2219} C_DIS
LIN {X 20.716,Y 119.9964,Z 137,A 76.4911,B 24.344,C -1.6777,E1 24.4247,E2 729.7728} C_DIS
LIN {X 17.7313,Y 120.4728,Z 137,A 78.0355,B 24.3436,C -1.6837,E1 24.4204,E2 728.2152} C_DIS
LIN {X 14.9026,Y 120.8552,Z 137,A 79.3078,B 24.3438,C -1.6808,E1 24.4169,E2 726.9511} C_DIS
LIN {X 11.792,Y 121.1974,Z 137,A 80.6941,B 24.344,C -1.6771,E1 24.4131,E2 725.5746} C_DIS
LIN {X 8.962,Y 121.4395,Z 137,A 82.0916,B 24.3438,C -1.6799,E1 24.4092,E2 724.1709} C_DIS
LIN {X 5.1001,Y 121.6634,Z 137,A 83.9715,B 24.3437,C -1.6826,E1 24.4039,E2 722.2853} C_DIS
LIN {X 1.4938,Y 121.7618,Z 137,A 85.6123,B 24.3439,C -1.6798,E1 24.3993,E2 720.6515} C_DIS
LIN {X -1.4905,Y 121.7618,Z 137,A 87.0055,B 24.3439,C -1.679,E1 24.3954,E2 719.2602} C_DIS
LIN {X -4.4748,Y 121.6878,Z 137,A 88.4005,B 24.3439,C -1.6782,E1 24.3916,E2 717.867} C_DIS
LIN {X -8.3038,Y 121.4875,Z 137,A 90.3653,B 24.3435,C -1.6847,E1 24.386,E2 715.8857} C_DIS
LIN {X -11.9348,Y 121.1837,Z 137,A 91.9199,B 24.3441,C -1.6767,E1 24.3818,E2 714.3497} C_DIS
LIN {X -15.4759,Y 120.7827,Z 137,A 93.4255,B 24.3446,C -1.6681,E1 24.3776,E2 712.8641} C_DIS
LIN {X -17.8622,Y 120.4541,Z 137,A 94.7866,B 24.344,C -1.6775,E1 24.3738,E2 711.479} C_DIS
LIN {X -20.8519,Y 119.9724,Z 137,A 96.2169,B 24.344,C -1.6767,E1 24.3699,E2 710.0492} C_DIS
LIN {X -23.8635,Y 119.4091,Z 137,A 97.5933,B 24.3443,C -1.6726,E1 24.3661,E2 708.6811} C_DIS
LIN {X -26.5611,Y 118.8387,Z 137,A 98.8668,B 24.3445,C -1.6704,E1 24.3627,E2 707.4113} C_DIS
LIN {X -29.3022,Y 118.1932,Z 137,A 100.3679,B 24.344,C -1.677,E1 24.3585,E2 705.8922} C_DIS
LIN {X -33.433,Y 117.0917,Z 137,A 102.4226,B 24.344,C -1.6768,E1 24.353,E2 703.8347} C_DIS
LIN {X -36.7701,Y 116.0854,Z 137,A 103.8884,B 24.3447,C -1.6672,E1 24.3491,E2 702.3895} C_DIS
LIN {X -39.739,Y 115.1026,Z 137,A 105.3221,B 24.3449,C -1.6638,E1 24.3454,E2 700.9614} C_DIS
LIN {X -43.0301,Y 113.9135,Z 137,A 107.0247,B 24.3449,C -1.6641,E1 24.3409,E2 699.2545} C_DIS
LIN {X -46.5982,Y 112.5011,Z 137,A 108.876,B 24.3449,C -1.6636,E1 24.3361,E2 697.4002} C_DIS
LIN {X -49.3593,Y 111.3174,Z 137,A 110.2795,B 24.3451,C -1.661,E1 24.3325,E2 695.9995} C_DIS
LIN {X -52.1696,Y 110.0282,Z 137,A 111.6918,B 24.3453,C -1.6569,E1 24.329,E2 694.5935} C_DIS
LIN {X -54.8821,Y 108.7008,Z 137,A 113.124,B 24.3454,C -1.6551,E1 24.3254,E2 693.1619} C_DIS
LIN {X -57.4,Y 107.3942,Z 137,A 114.4648,B 24.3456,C -1.6531,E1 24.3221,E2 691.8221} C_DIS
LIN {X -60.1363,Y 105.8861,Z 137,A 115.9044,B 24.3458,C -1.6492,E1 24.3186,E2 690.3878} C_DIS
LIN {X -62.7081,Y 104.384,Z 137,A 117.3519,B 24.3458,C -1.6486,E1 24.3151,E2 688.9371} C_DIS
LIN {X -65.1259,Y 102.8924,Z 137,A 118.8584,B 24.3455,C -1.6535,E1 24.3115,E2 687.4139} C_DIS
LIN {X -68.8945,Y 100.4079,Z 137,A 120.8582,B 24.3462,C -1.6439,E1 24.3069,E2 685.4305} C_DIS
LIN {X -71.4517,Y 98.6045,Z 137,A 122.3057,B 24.3464,C -1.6398,E1 24.3036,E2 683.9879} C_DIS
LIN {X -74.3809,Y 96.4145,Z 137,A 124.1884,B 24.3462,C -1.6431,E1 24.2994,E2 682.09} C_DIS
LIN {X -77.9296,Y 93.5697,Z 137,A 126.3428,B 24.3465,C -1.639,E1 24.2947,E2 679.9372} C_DIS
LIN {X -81.277,Y 90.6766,Z 137,A 128.4199,B 24.3468,C -1.6341,E1 24.2904,E2 677.8638} C_DIS
LIN {X -84.5027,Y 87.6788,Z 137,A 130.5137,B 24.347,C -1.6301,E1 24.2861,E2 675.7708} C_DIS
LIN {X -87.6774,Y 84.5041,Z 137,A 132.5026,B 24.3477,C -1.6196,E1 24.2823,E2 673.7989} C_DIS
LIN {X -90.2276,Y 81.7752,Z 137,A 134.4117,B 24.3476,C -1.6216,E1 24.2786,E2 671.876} C_DIS
LIN {X -93.1722,Y 78.4039,Z 137,A 136.5243,B 24.3479,C -1.6164,E1 24.2748,E2 669.7663} C_DIS
LIN {X -95.9993,Y 74.9164,Z 137,A 138.5038,B 24.3486,C -1.6051,E1 24.2714,E2 667.8048} C_DIS
LIN {X -97.808,Y 72.5386,Z 137,A 139.9142,B 24.3488,C -1.6015,E1 24.269,E2 666.3962} C_DIS
LIN {X -99.556,Y 70.1199,Z 137,A 141.3612,B 24.3489,C -1.5994,E1 24.2667,E2 664.9469} C_DIS
LIN {X -101.2671,Y 67.6252,Z 137,A 142.7829,B 24.3492,C -1.5954,E1 24.2645,E2 663.5279} C_DIS
LIN {X -103.2313,Y 64.5879,Z 137,A 144.6389,B 24.3491,C -1.5971,E1 24.2617,E2 661.6581} C_DIS
LIN {X -105.1875,Y 61.3509,Z 137,A 146.2885,B 24.3497,C -1.5864,E1 24.2594,E2 660.0258} C_DIS
LIN {X -106.7045,Y 58.6727,Z 137,A 147.7415,B 24.35,C -1.5823,E1 24.2574,E2 658.5748} C_DIS
LIN {X -108.0902,Y 56.0769,Z 137,A 149.1169,B 24.3503,C -1.5778,E1 24.2556,E2 657.2028} C_DIS
LIN {X -109.4409,Y 53.3921,Z 137,A 150.5372,B 24.3505,C -1.5739,E1 24.2538,E2 655.7844} C_DIS
LIN {X -110.7744,Y 50.5681,Z 137,A 152.0095,B 24.3508,C -1.5695,E1 24.2521,E2 654.3144} C_DIS
LIN {X -111.9775,Y 47.8442,Z 137,A 153.4153,B 24.351,C -1.5654,E1 24.2506,E2 652.9106} C_DIS
LIN {X -113.0606,Y 45.2235,Z 137,A 154.7673,B 24.3512,C -1.5621,E1 24.2491,E2 651.559} C_DIS
LIN {X -114.3487,Y 41.863,Z 137,A 156.6887,B 24.351,C -1.5664,E1 24.2472,E2 649.6159} C_DIS
LIN {X -115.8488,Y 37.511,Z 137,A 158.8515,B 24.3514,C -1.5595,E1 24.2453,E2 647.4574} C_DIS
LIN {X -116.9518,Y 33.9142,Z 137,A 160.5552,B 24.3519,C -1.551,E1 24.244,E2 645.7642} C_DIS
LIN {X -117.7859,Y 30.8952,Z 137,A 161.9151,B 24.3524,C -1.5415,E1 24.243,E2 644.4194} C_DIS
LIN {X -118.5079,Y 27.9999,Z 137,A 163.319,B 24.3527,C -1.537,E1 24.2421,E2 643.018} C_DIS
LIN {X -119.1327,Y 25.2083,Z 137,A 164.6814,B 24.3529,C -1.5333,E1 24.2413,E2 641.6562} C_DIS
LIN {X -119.8032,Y 21.7975,Z 137,A 166.2056,B 24.3535,C -1.5234,E1 24.2405,E2 640.1471} C_DIS
LIN {X -120.2469,Y 19.2054,Z 137,A 167.5919,B 24.3534,C -1.5256,E1 24.2399,E2 638.7468} C_DIS
LIN {X -120.6616,Y 16.3998,Z 137,A 168.9677,B 24.3535,C -1.523,E1 24.2393,E2 637.369} C_DIS
LIN {X -121.0436,Y 13.2802,Z 137,A 170.4198,B 24.3539,C -1.5171,E1 24.2389,E2 635.9224} C_DIS
LIN {X -121.3912,Y 9.6148,Z 137,A 172.4266,B 24.3535,C -1.523,E1 24.2384,E2 633.8887} C_DIS
LIN {X -121.6301,Y 5.8359,Z 137,A 173.9421,B 24.3545,C -1.506,E1 24.2381,E2 632.4055} C_DIS
LIN {X -121.7395,Y 2.7818,Z 137,A 175.4006,B 24.3548,C -1.5021,E1 24.2381,E2 630.9472} C_DIS
LIN {X -121.7731,Y -0.0347,Z 137,A 176.8148,B 24.3548,C -1.5015,E1 24.2381,E2 629.5258} C_DIS
LIN {X -121.7209,Y -3.4496,Z 137,A 178.3585,B 24.3552,C -1.4937,E1 24.2381,E2 627.9916} C_DIS
LIN {X -121.6235,Y -5.9679,Z 137,A 179.5819,B 24.3554,C -1.4914,E1 24.2383,E2 626.7661} C_DIS
LIN {X -121.4312,Y -9.075,Z 137,A -179.0022,B 24.3558,C -1.4846,E1 24.2385,E2 625.3581} C_DIS
LIN {X -121.188,Y -11.8902,Z 137,A -177.6285,B 24.3559,C -1.4822,E1 24.2389,E2 623.9818} C_DIS
LIN {X -120.8074,Y -15.2875,Z 137,A -176.1027,B 24.3564,C -1.4735,E1 24.2394,E2 622.4678} C_DIS
LIN {X -120.4541,Y -17.8618,Z 137,A -174.7969,B 24.3564,C -1.4731,E1 24.2399,E2 621.1549} C_DIS
LIN {X -119.982,Y -20.7988,Z 137,A -173.2221,B 24.3563,C -1.4761,E1 24.2406,E2 619.5633} C_DIS
LIN {X -119.4024,Y -23.8962,Z 137,A -171.873,B 24.3568,C -1.4658,E1 24.2413,E2 618.2312} C_DIS
LIN {X -118.8108,Y -26.6832,Z 137,A -170.5253,B 24.3571,C -1.4619,E1 24.2422,E2 616.8848} C_DIS
LIN {X -118.1209,Y -29.587,Z 137,A -169.073,B 24.3571,C -1.4595,E1 24.2431,E2 615.4295} C_DIS
LIN {X -117.3205,Y -32.6148,Z 137,A -167.5834,B 24.3574,C -1.4557,E1 24.2442,E2 613.9404} C_DIS
LIN {X -116.356,Y -35.9046,Z 137,A -166.1332,B 24.3581,C -1.4438,E1 24.2454,E2 612.5105} C_DIS
LIN {X -115.6233,Y -38.1984,Z 137,A -164.8298,B 24.3579,C -1.4476,E1 24.2465,E2 611.1901} C_DIS
LIN {X -114.6518,Y -41.0223,Z 137,A -163.3524,B 24.3579,C -1.4465,E1 24.2479,E2 609.7068} C_DIS
LIN {X -113.5543,Y -43.9682,Z 137,A -161.8912,B 24.3582,C -1.4414,E1 24.2493,E2 608.2498} C_DIS
LIN {X -112.013,Y -47.7621,Z 137,A -159.9536,B 24.3585,C -1.4362,E1 24.2514,E2 606.3138} C_DIS
LIN {X -110.6566,Y -50.8228,Z 137,A -158.4371,B 24.3589,C -1.4291,E1 24.2531,E2 604.8059} C_DIS
LIN {X -109.1615,Y -53.9586,Z 137,A -156.9266,B 24.3594,C -1.4192,E1 24.255,E2 603.3112} C_DIS
LIN {X -108.0212,Y -56.2082,Z 137,A -155.6847,B 24.3594,C -1.4182,E1 24.2565,E2 602.0649} C_DIS
LIN {X -106.6827,Y -58.7121,Z 137,A -154.2212,B 24.3594,C -1.42,E1 24.2585,E2 600.5891} C_DIS
LIN {X -104.7719,Y -62.0578,Z 137,A -152.2687,B 24.3594,C -1.4211,E1 24.2613,E2 598.6235} C_DIS
LIN {X -102.8759,Y -65.152,Z 137,A -150.6912,B 24.3599,C -1.4109,E1 24.2636,E2 597.0624} C_DIS
LIN {X -100.8429,Y -68.2562,Z 137,A -148.8167,B 24.3599,C -1.412,E1 24.2665,E2 595.1758} C_DIS
LIN {X -98.6055,Y -71.4504,Z 137,A -147.1172,B 24.3604,C -1.4015,E1 24.2692,E2 593.4933} C_DIS
LIN {X -96.4154,Y -74.3797,Z 137,A -145.2289,B 24.3602,C -1.4045,E1 24.2724,E2 591.5884} C_DIS
LIN {X -93.6546,Y -77.8271,Z 137,A -143.2934,B 24.3608,C -1.3933,E1 24.2758,E2 589.6707} C_DIS
LIN {X -91.2332,Y -80.6517,Z 137,A -141.4637,B 24.3608,C -1.3927,E1 24.2792,E2 587.8341} C_DIS
LIN {X -88.6601,Y -83.4721,Z 137,A -139.6256,B 24.361,C -1.3905,E1 24.2827,E2 585.993} C_DIS
LIN {X -86.1039,Y -86.1073,Z 137,A -137.8261,B 24.361,C -1.3899,E1 24.2862,E2 584.1871} C_DIS
LIN {X -82.8154,Y -89.2741,Z 137,A -135.6693,B 24.3612,C -1.3859,E1 24.2906,E2 582.0311} C_DIS
LIN {X -79.4922,Y -92.2452,Z 137,A -133.5959,B 24.3615,C -1.3806,E1 24.295,E2 579.9619} C_DIS
LIN {X -76.1246,Y -95.0441,Z 137,A -131.4925,B 24.3616,C -1.3786,E1 24.2995,E2 577.8553} C_DIS
LIN {X -72.5332,Y -97.812,Z 137,A -129.5168,B 24.3622,C -1.3679,E1 24.3039,E2 575.8985} C_DIS
LIN {X -70.1188,Y -99.5568,Z 137,A -128.0006,B 24.362,C -1.3705,E1 24.3073,E2 574.3704} C_DIS
LIN {X -66.6026,Y -101.9432,Z 137,A -126.0425,B 24.3623,C -1.3654,E1 24.3119,E2 572.418} C_DIS
LIN {X -63.8731,Y -103.6749,Z 137,A -124.546,B 24.3625,C -1.362,E1 24.3154,E2 570.925} C_DIS
LIN {X -61.314,Y -105.2089,Z 137,A -123.1346,B 24.3625,C -1.3603,E1 24.3188,E2 569.5135} C_DIS
LIN {X -58.5718,Y -106.7597,Z 137,A -121.7176,B 24.3628,C -1.3553,E1 24.3222,E2 568.1042} C_DIS
LIN {X -56.0857,Y -108.0855,Z 137,A -120.3488,B 24.3628,C -1.3555,E1 24.3256,E2 566.7312} C_DIS
LIN {X -53.4199,Y -109.4272,Z 137,A -118.9426,B 24.3629,C -1.3539,E1 24.3292,E2 565.3252} C_DIS
LIN {X -50.0421,Y -111.012,Z 137,A -117.0268,B 24.3627,C -1.359,E1 24.3341,E2 563.3919} C_DIS
LIN {X -46.5938,Y -112.5029,Z 137,A -115.4144,B 24.3631,C -1.3502,E1 24.3382,E2 561.7973} C_DIS
LIN {X -43.6899,Y -113.6625,Z 137,A -113.9398,B 24.3631,C -1.3489,E1 24.342,E2 560.3226} C_DIS
LIN {X -40.6708,Y -114.7785,Z 137,A -112.4296,B 24.3633,C -1.3473,E1 24.346,E2 558.813} C_DIS
LIN {X -38.0662,Y -115.6673,Z 137,A -111.1419,B 24.3633,C -1.3459,E1 24.3494,E2 557.5262} C_DIS
LIN {X -35.2208,Y -116.5653,Z 137,A -109.6826,B 24.3633,C -1.3474,E1 24.3533,E2 556.0608} C_DIS
LIN {X -31.1781,Y -117.7105,Z 137,A -107.7072,B 24.3633,C -1.346,E1 24.3586,E2 554.0854} C_DIS
LIN {X -28.0111,Y -118.5051,Z 137,A -106.2102,B 24.3635,C -1.3434,E1 24.3627,E2 552.5927} C_DIS
LIN {X -25.2792,Y -119.1174,Z 137,A -104.7205,B 24.3631,C -1.3506,E1 24.3668,E2 551.0836} C_DIS
LIN {X -22.1526,Y -119.7397,Z 137,A -103.2091,B 24.3631,C -1.3506,E1 24.3709,E2 549.5707} C_DIS
LIN {X -18.4412,Y -120.3652,Z 137,A -101.5167,B 24.3633,C -1.3465,E1 24.3756,E2 547.8866} C_DIS
LIN {X -14.9071,Y -120.8547,Z 137,A -99.8781,B 24.3634,C -1.3443,E1 24.3801,E2 546.2521} C_DIS
LIN {X -11.7965,Y -121.197,Z 137,A -98.3526,B 24.3633,C -1.3466,E1 24.3844,E2 544.7201} C_DIS
LIN {X -7.6138,Y -121.5315,Z 137,A -96.429,B 24.3634,C -1.3442,E1 24.3897,E2 542.8015} C_DIS
LIN {X -4.3359,Y -121.6932,Z 137,A -94.9573,B 24.3636,C -1.341,E1 24.3938,E2 541.3373} C_DIS
LIN {X -1.4972,Y -121.7617,Z 137,A -93.5747,B 24.3635,C -1.3434,E1 24.3977,E2 539.9489} C_DIS
LIN {X 0.8692,Y -121.766,Z 137,A -92.8303,B 24.3643,C -1.3266,E1 24.3996,E2 539.2452} C_DIS
Enddeposition()
LIN {X 0.9001,Y -127.1293,Z 138,A -93.1611,B 24.9659,C -1.3489,E1 25.0004,E2 539.6053} C_DIS
Startdeposition()
$VEL.CP = VEL_PRINT
LIN {X 4.8588,Y -127.0398,Z 138,A -90.6899,B 24.9641,C -1.3837,E1 25.0075,E2 537.0522} C_DIS
LIN {X 8.5356,Y -126.8478,Z 138,A -88.9379,B 24.9639,C -1.389,E1 25.0125,E2 535.2882} C_DIS
LIN {X 12.1443,Y -126.5512,Z 138,A -87.524,B 24.9644,C -1.3789,E1 25.0163,E2 533.8991} C_DIS
LIN {X 16.3288,Y -126.0796,Z 138,A -85.5753,B 24.9642,C -1.3826,E1 25.0217,E2 531.943} C_DIS
LIN {X 18.7801,Y -125.7395,Z 138,A -84.3214,B 24.9638,C -1.3904,E1 25.0253,E2 530.6719} C_DIS
LIN {X 22.1313,Y -125.1916,Z 138,A -82.886,B 24.964,C -1.3868,E1 25.0292,E2 529.2464} C_DIS
LIN {X 25.084,Y -124.6335,Z 138,A -81.5618,B 24.964,C -1.3865,E1 25.0328,E2 527.9247} C_DIS
LIN {X 28.0949,Y -123.9893,Z 138,A -80.2813,B 24.9642,C -1.3823,E1 25.0363,E2 526.6556} C_DIS
LIN {X 30.6901,Y -123.3738,Z 138,A -78.8761,B 24.9636,C -1.3938,E1 25.0401,E2 525.2252} C_DIS
LIN {X 34.0322,Y -122.4927,Z 138,A -77.4331,B 24.9638,C -1.3897,E1 25.044,E2 523.7943} C_DIS
LIN {X 37.0117,Y -121.6256,Z 138,A -76.163,B 24.9641,C -1.3848,E1 25.0474,E2 522.538} C_DIS
LIN {X 39.4266,Y -120.8667,Z 138,A -74.7285,B 24.9632,C -1.4012,E1 25.0513,E2 521.0675} C_DIS
LIN {X 42.3823,Y -119.8622,Z 138,A -73.4761,B 24.9635,C -1.3951,E1 25.0545,E2 519.832} C_DIS
LIN {X 45.5485,Y -118.6938,Z 138,A -71.8722,B 24.9632,C -1.4014,E1 25.0588,E2 518.2165} C_DIS
LIN {X 48.4283,Y -117.5485,Z 138,A -70.4666,B 24.9631,C -1.4039,E1 25.0624,E2 516.8082} C_DIS
LIN {X 51.4733,Y -116.2467,Z 138,A -69.2029,B 24.9636,C -1.3944,E1 25.0656,E2 515.57} C_DIS
LIN {X 54.5443,Y -114.8371,Z 138,A -67.5357,B 24.9631,C -1.4043,E1 25.0698,E2 513.8837} C_DIS
LIN {X 57.4234,Y -113.4248,Z 138,A -66.2528,B 24.9634,C -1.3984,E1 25.073,E2 512.6183} C_DIS
LIN {X 60.5257,Y -111.8027,Z 138,A -64.4053,B 24.9625,C -1.415,E1 25.0776,E2 510.7367} C_DIS
LIN {X 64.2689,Y -109.6931,Z 138,A -62.5125,B 24.9625,C -1.4163,E1 25.0822,E2 508.8465} C_DIS
LIN {X 67.7346,Y -107.5876,Z 138,A -60.6908,B 24.9623,C -1.4196,E1 25.0865,E2 507.023} C_DIS
LIN {X 71.4324,Y -105.1689,Z 138,A -58.7061,B 24.9621,C -1.4232,E1 25.0912,E2 505.0362} C_DIS
LIN {X 74.9706,Y -102.6771,Z 138,A -56.8043,B 24.962,C -1.4248,E1 25.0955,E2 503.1374} C_DIS
LIN {X 78.2075,Y -100.2337,Z 138,A -54.9164,B 24.9616,C -1.4319,E1 25.0997,E2 501.2395} C_DIS
LIN {X 81.5028,Y -97.5726,Z 138,A -53.0471,B 24.9615,C -1.4342,E1 25.1037,E2 499.3721} C_DIS
LIN {X 84.6425,Y -94.8617,Z 138,A -51.1604,B 24.9612,C -1.4395,E1 25.1077,E2 497.4803} C_DIS
LIN {X 87.9288,Y -91.8236,Z 138,A -49.2136,B 24.9612,C -1.4407,E1 25.1116,E2 495.5387} C_DIS
LIN {X 90.9728,Y -88.8092,Z 138,A -47.2603,B 24.9608,C -1.4467,E1 25.1155,E2 493.5795} C_DIS
LIN {X 93.8762,Y -85.7348,Z 138,A -45.3323,B 24.9605,C -1.4528,E1 25.1191,E2 491.6457} C_DIS
LIN {X 96.5984,Y -82.6556,Z 138,A -43.4825,B 24.9602,C -1.4575,E1 25.1225,E2 489.793} C_DIS
LIN {X 99.38,Y -79.2886,Z 138,A -41.5518,B 24.96,C -1.4609,E1 25.1259,E2 487.8634} C_DIS
LIN {X 102.1164,Y -75.732,Z 138,A -39.5603,B 24.9598,C -1.4648,E1 25.1293,E2 485.8721} C_DIS
LIN {X 104.5921,Y -72.2752,Z 138,A -37.6207,B 24.9594,C -1.4714,E1 25.1324,E2 483.9263} C_DIS
LIN {X 106.9751,Y -68.698,Z 138,A -35.7153,B 24.9592,C -1.4753,E1 25.1353,E2 482.0212} C_DIS
LIN {X 109.2235,Y -65.0637,Z 138,A -33.8259,B 24.959,C -1.4791,E1 25.138,E2 480.1327} C_DIS
LIN {X 111.4167,Y -61.2334,Z 138,A -31.8125,B 24.9586,C -1.4863,E1 25.1408,E2 478.1128} C_DIS
LIN {X 113.1648,Y -57.9342,Z 138,A -30.239,B 24.9586,C -1.4856,E1 25.1428,E2 476.5491} C_DIS
LIN {X 114.4605,Y -55.3326,Z 138,A -28.8753,B 24.9583,C -1.4924,E1 25.1445,E2 475.1767} C_DIS
LIN {X 115.9353,Y -52.1696,Z 138,A -27.6048,B 24.9589,C -1.4813,E1 25.1459,E2 473.9394} C_DIS
LIN {X 117.2026,Y -49.2566,Z 138,A -26.1588,B 24.9586,C -1.4865,E1 25.1476,E2 472.489} C_DIS
LIN {X 118.3911,Y -46.3273,Z 138,A -24.5335,B 24.9578,C -1.5016,E1 25.1493,E2 470.837} C_DIS
LIN {X 119.5243,Y -43.3196,Z 138,A -23.1345,B 24.9576,C -1.5035,E1 25.1506,E2 469.4413} C_DIS
LIN {X 120.5319,Y -40.4319,Z 138,A -21.7488,B 24.9574,C -1.5083,E1 25.1519,E2 468.0521} C_DIS
LIN {X 121.4793,Y -37.4898,Z 138,A -20.5155,B 24.9576,C -1.5043,E1 25.1529,E2 466.8352} C_DIS
LIN {X 122.3793,Y -34.4378,Z 138,A -19.0802,B 24.9573,C -1.509,E1 25.154,E2 465.3971} C_DIS
LIN {X 123.1759,Y -31.4699,Z 138,A -17.6046,B 24.9568,C -1.5183,E1 25.1551,E2 463.9081} C_DIS
LIN {X 123.8492,Y -28.7086,Z 138,A -16.4128,B 24.9568,C -1.5177,E1 25.1558,E2 462.7246} C_DIS
LIN {X 124.4289,Y -26.0893,Z 138,A -14.9483,B 24.9558,C -1.5352,E1 25.1567,E2 461.2273} C_DIS
LIN {X 125.0334,Y -23.0148,Z 138,A -13.5976,B 24.9558,C -1.5366,E1 25.1574,E2 459.8813} C_DIS
LIN {X 125.5945,Y -19.7167,Z 138,A -12.3147,B 24.9562,C -1.5296,E1 25.158,E2 458.6224} C_DIS
LIN {X 126.0393,Y -16.6367,Z 138,A -10.8437,B 24.9557,C -1.5379,E1 25.1585,E2 457.1406} C_DIS
LIN {X 126.3398,Y -14.1868,Z 138,A -9.6321,B 24.9552,C -1.5468,E1 25.1589,E2 455.9152} C_DIS
LIN {X 126.6861,Y -10.6448,Z 138,A -8.105,B 24.9552,C -1.548,E1 25.1593,E2 454.3943} C_DIS
LIN {X 126.947,Y -6.8848,Z 138,A -6.3361,B 24.9546,C -1.5573,E1 25.1596,E2 452.6139} C_DIS
LIN {X 127.0831,Y -3.548,Z 138,A -4.9161,B 24.9546,C -1.5578,E1 25.1598,E2 451.2012} C_DIS
LIN {X 127.1363,Y 0.0168,Z 138,A -3.1877,B 24.9538,C -1.5695,E1 25.1598,E2 449.4556} C_DIS
LIN {X 127.0765,Y 3.7872,Z 138,A -1.5259,B 24.9536,C -1.5731,E1 25.1597,E2 447.7951} C_DIS
LIN {X 126.9079,Y 7.559,Z 138,A 0.0901,B 24.9536,C -1.5741,E1 25.1594,E2 446.1864} C_DIS
LIN {X 126.6919,Y 10.5761,Z 138,A 1.405,B 24.9535,C -1.576,E1 25.1591,E2 444.8748} C_DIS
LIN {X 126.3245,Y 14.3297,Z 138,A 3.231,B 24.9527,C -1.5882,E1 25.1586,E2 443.0308} C_DIS
LIN {X 125.8916,Y 17.721,Z 138,A 4.4609,B 24.9534,C -1.5767,E1 25.1582,E2 441.8353} C_DIS
LIN {X 125.4353,Y 20.7049,Z 138,A 5.9381,B 24.9528,C -1.5873,E1 25.1575,E2 440.3418} C_DIS
LIN {X 124.9688,Y 23.3605,Z 138,A 7.2325,B 24.9523,C -1.5954,E1 25.1568,E2 439.036} C_DIS
LIN {X 124.3266,Y 26.5632,Z 138,A 8.6578,B 24.9522,C -1.5976,E1 25.156,E2 437.6138} C_DIS
LIN {X 123.6926,Y 29.376,Z 138,A 9.9916,B 24.9518,C -1.6035,E1 25.1552,E2 436.2738} C_DIS
LIN {X 122.9107,Y 32.491,Z 138,A 11.3569,B 24.9518,C -1.6037,E1 25.1542,E2 434.9159} C_DIS
LIN {X 122.0881,Y 35.4568,Z 138,A 12.7369,B 24.9516,C -1.6076,E1 25.1532,E2 433.5345} C_DIS
LIN {X 121.3396,Y 37.9462,Z 138,A 13.9636,B 24.9512,C -1.6141,E1 25.1522,E2 432.2995} C_DIS
LIN {X 120.2103,Y 41.3783,Z 138,A 15.3214,B 24.9517,C -1.6049,E1 25.151,E2 430.9712} C_DIS
LIN {X 119.3306,Y 43.8569,Z 138,A 16.8453,B 24.9504,C -1.6262,E1 25.1495,E2 429.4054} C_DIS
LIN {X 118.0191,Y 47.2668,Z 138,A 18.3723,B 24.9505,C -1.6249,E1 25.148,E2 427.8901} C_DIS
LIN {X 116.8054,Y 50.1912,Z 138,A 19.5552,B 24.9511,C -1.6163,E1 25.1467,E2 426.7339} C_DIS
LIN {X 115.5078,Y 53.1092,Z 138,A 21.188,B 24.9502,C -1.6306,E1 25.1448,E2 425.0762} C_DIS
LIN {X 114.0973,Y 56.0751,Z 138,A 22.5589,B 24.9502,C -1.6291,E1 25.1432,E2 423.7161} C_DIS
LIN {X 112.6855,Y 58.861,Z 138,A 24.0584,B 24.9497,C -1.6379,E1 25.1412,E2 422.2039} C_DIS
LIN {X 110.7569,Y 62.4178,Z 138,A 25.9151,B 24.9493,C -1.6447,E1 25.1387,E2 420.3409} C_DIS
LIN {X 108.8513,Y 65.6845,Z 138,A 27.6657,B 24.9489,C -1.6518,E1 25.1362,E2 418.5827} C_DIS
LIN {X 106.4826,Y 69.4591,Z 138,A 29.6593,B 24.9486,C -1.6563,E1 25.1332,E2 416.5882} C_DIS
LIN {X 104.1259,Y 72.9453,Z 138,A 31.5276,B 24.9484,C -1.6598,E1 25.1302,E2 414.721} C_DIS
LIN {X 101.7267,Y 76.2554,Z 138,A 33.4184,B 24.9479,C -1.6669,E1 25.1271,E2 412.8224} C_DIS
LIN {X 99.2165,Y 79.4941,Z 138,A 35.2565,B 24.9477,C -1.671,E1 25.1239,E2 410.9833} C_DIS
LIN {X 96.554,Y 82.7072,Z 138,A 37.1029,B 24.9475,C -1.6737,E1 25.1206,E2 409.1389} C_DIS
LIN {X 93.8762,Y 85.7348,Z 138,A 38.9414,B 24.9472,C -1.6788,E1 25.1171,E2 407.2966} C_DIS
LIN {X 91.0251,Y 88.7559,Z 138,A 40.8242,B 24.9469,C -1.6835,E1 25.1135,E2 405.4108} C_DIS
LIN {X 88.0469,Y 91.7108,Z 138,A 42.6836,B 24.9467,C -1.686,E1 25.1098,E2 403.5534} C_DIS
LIN {X 84.9297,Y 94.6044,Z 138,A 44.5684,B 24.9466,C -1.6883,E1 25.1059,E2 401.6708} C_DIS
LIN {X 81.602,Y 97.4893,Z 138,A 46.4831,B 24.9466,C -1.6886,E1 25.1018,E2 399.7628} C_DIS
LIN {X 78.4241,Y 100.0636,Z 138,A 48.3206,B 24.9464,C -1.6918,E1 25.0978,E2 397.9246} C_DIS
LIN {X 75.1507,Y 102.5448,Z 138,A 50.1615,B 24.9462,C -1.6946,E1 25.0937,E2 396.0837} C_DIS
LIN {X 72.0598,Y 104.7399,Z 138,A 51.9274,B 24.9458,C -1.7005,E1 25.0896,E2 394.31} C_DIS
LIN {X 68.4169,Y 107.155,Z 138,A 53.8503,B 24.9458,C -1.7013,E1 25.0852,E2 392.3914} C_DIS
LIN {X 64.7434,Y 109.4143,Z 138,A 55.8475,B 24.9454,C -1.707,E1 25.0804,E2 390.3871} C_DIS
LIN {X 61.1904,Y 111.4401,Z 138,A 57.7048,B 24.9452,C -1.7103,E1 25.0758,E2 388.5273} C_DIS
LIN {X 57.9342,Y 113.1648,Z 138,A 59.0079,B 24.9462,C -1.6945,E1 25.0727,E2 387.2653} C_DIS
LIN {X 55.1251,Y 114.5597,Z 138,A 60.6418,B 24.9454,C -1.7074,E1 25.0685,E2 385.6051} C_DIS
LIN {X 52.104,Y 115.9646,Z 138,A 62.0697,B 24.9454,C -1.7055,E1 25.0649,E2 384.1854} C_DIS
LIN {X 49.2566,Y 117.2026,Z 138,A 63.4156,B 24.9456,C -1.7043,E1 25.0615,E2 382.8454} C_DIS
LIN {X 46.3273,Y 118.3911,Z 138,A 64.9335,B 24.9452,C -1.7105,E1 25.0575,E2 381.3163} C_DIS
LIN {X 43.3665,Y 119.5074,Z 138,A 66.32,B 24.9452,C -1.7099,E1 25.0539,E2 379.9342} C_DIS
LIN {X 40.4319,Y 120.5319,Z 138,A 67.7515,B 24.945,C -1.7126,E1 25.0501,E2 378.4991} C_DIS
LIN {X 37.3341,Y 121.5269,Z 138,A 69.0246,B 24.9456,C -1.7042,E1 25.0468,E2 377.2483} C_DIS
LIN {X 34.9821,Y 122.2271,Z 138,A 70.4543,B 24.9445,C -1.7211,E1 25.0429,E2 375.781} C_DIS
LIN {X 31.5413,Y 123.1578,Z 138,A 71.9451,B 24.9448,C -1.7164,E1 25.0389,E2 374.3037} C_DIS
LIN {X 28.9694,Y 123.7896,Z 138,A 73.0751,B 24.945,C -1.7139,E1 25.0358,E2 373.1813} C_DIS
LIN {X 25.6061,Y 124.5273,Z 138,A 74.6534,B 24.9448,C -1.716,E1 25.0315,E2 371.5999} C_DIS
LIN {X 22.797,Y 125.0724,Z 138,A 75.8052,B 24.9452,C -1.7097,E1 25.0284,E2 370.4644} C_DIS
LIN {X 19.6928,Y 125.5982,Z 138,A 77.2783,B 24.945,C -1.7129,E1 25.0243,E2 368.9853} C_DIS
LIN {X 16.7832,Y 126.0201,Z 138,A 78.7178,B 24.9446,C -1.7188,E1 25.0203,E2 367.5329} C_DIS
LIN {X 13.6731,Y 126.3951,Z 138,A 80.0399,B 24.9449,C -1.7147,E1 25.0167,E2 366.2216} C_DIS
LIN {X 11.2655,Y 126.6337,Z 138,A 81.3039,B 24.9443,C -1.7233,E1 25.0131,E2 364.9378} C_DIS
LIN {X 7.9364,Y 126.8847,Z 138,A 82.6422,B 24.9449,C -1.7152,E1 25.0094,E2 363.6194} C_DIS
LIN {X 3.7311,Y 127.078,Z 138,A 84.5736,B 24.9448,C -1.7168,E1 25.004,E2 361.6849} C_DIS
LIN {X 0.6531,Y 127.131,Z 138,A 86.0423,B 24.9445,C -1.7205,E1 24.9999,E2 360.2074} C_DIS
LIN {X -2.8219,Y 127.1033,Z 138,A 87.6863,B 24.9443,C -1.7239,E1 24.9953,E2 358.5553} C_DIS
LIN {X -6.0131,Y 126.9908,Z 138,A 89.0039,B 24.9447,C -1.7175,E1 24.9916,E2 357.2525} C_DIS
LIN {X -9.3288,Y 126.7898,Z 138,A 90.4263,B 24.945,C -1.7133,E1 24.9877,E2 355.8397} C_DIS
LIN {X -11.892,Y 126.5754,Z 138,A 91.6345,B 24.9449,C -1.7151,E1 24.9843,E2 354.6266} C_DIS
LIN {X -14.4008,Y 126.316,Z 138,A 92.8917,B 24.9445,C -1.7203,E1 24.9808,E2 353.3563} C_DIS
LIN {X -17.8752,Y 125.8696,Z 138,A 94.2135,B 24.9454,C -1.7069,E1 24.9772,E2 352.0653} C_DIS
LIN {X -20.6584,Y 125.443,Z 138,A 95.6427,B 24.945,C -1.7137,E1 24.9732,E2 350.6186} C_DIS
LIN {X -23.3705,Y 124.9669,Z 138,A 96.948,B 24.9448,C -1.7158,E1 24.9696,E2 349.3069} C_DIS
LIN {X -26.6968,Y 124.2978,Z 138,A 98.376,B 24.9452,C -1.7097,E1 24.9658,E2 347.8918} C_DIS
LIN {X -29.5952,Y 123.6398,Z 138,A 99.6905,B 24.9454,C -1.7072,E1 24.9622,E2 346.5815} C_DIS
LIN {X -32.5629,Y 122.8915,Z 138,A 101.1692,B 24.9452,C -1.7106,E1 24.9582,E2 345.0926} C_DIS
LIN {X -35.4673,Y 122.085,Z 138,A 102.501,B 24.9453,C -1.7078,E1 24.9546,E2 343.7652} C_DIS
LIN {X -39.4266,Y 120.8667,Z 138,A 104.5314,B 24.945,C -1.7134,E1 24.9492,E2 341.7179} C_DIS
LIN {X -42.5669,Y 119.7957,Z 138,A 105.7995,B 24.9458,C -1.7007,E1 24.9459,E2 340.4775} C_DIS
LIN {X -45.6943,Y 118.6372,Z 138,A 107.4262,B 24.9455,C -1.7046,E1 24.9416,E2 338.8382} C_DIS
LIN {X -48.263,Y 117.6176,Z 138,A 108.795,B 24.9453,C -1.7086,E1 24.938,E2 337.4568} C_DIS
LIN {X -51.6732,Y 116.1573,Z 138,A 110.1718,B 24.9463,C -1.6922,E1 24.9346,E2 336.1159} C_DIS
LIN {X -54.5443,Y 114.8371,Z 138,A 111.7488,B 24.946,C -1.6972,E1 24.9306,E2 334.523} C_DIS
LIN {X -57.419,Y 113.4271,Z 138,A 113.1092,B 24.9464,C -1.6909,E1 24.9272,E2 333.1739} C_DIS
LIN {X -60.5257,Y 111.8027,Z 138,A 114.9096,B 24.9459,C -1.6985,E1 24.9227,E2 331.3502} C_DIS
LIN {X -64.0454,Y 109.8244,Z 138,A 116.7301,B 24.9461,C -1.6953,E1 24.9183,E2 329.532} C_DIS
LIN {X -67.6505,Y 107.6407,Z 138,A 118.6446,B 24.9463,C -1.6924,E1 24.9138,E2 327.6185} C_DIS
LIN {X -71.4529,Y 105.155,Z 138,A 120.6751,B 24.9466,C -1.6876,E1 24.909,E2 325.5928} C_DIS
LIN {X -74.9396,Y 102.6998,Z 138,A 122.5921,B 24.9469,C -1.6833,E1 24.9047,E2 323.6791} C_DIS
LIN {X -78.2075,Y 100.2337,Z 138,A 124.5044,B 24.9469,C -1.6825,E1 24.9005,E2 321.7619} C_DIS
LIN {X -81.6128,Y 97.4803,Z 138,A 126.4446,B 24.9473,C -1.6765,E1 24.8963,E2 319.8285} C_DIS
LIN {X -84.9297,Y 94.6044,Z 138,A 128.3995,B 24.9477,C -1.6708,E1 24.8922,E2 317.8795} C_DIS
LIN {X -87.9479,Y 91.8054,Z 138,A 130.2928,B 24.9479,C -1.6682,E1 24.8884,E2 315.9847} C_DIS
LIN {X -91.0538,Y 88.7266,Z 138,A 132.3296,B 24.9479,C -1.6664,E1 24.8844,E2 313.9436} C_DIS
LIN {X -94.0978,Y 85.4907,Z 138,A 134.2805,B 24.9484,C -1.6589,E1 24.8807,E2 312.0019} C_DIS
LIN {X -96.9601,Y 82.2301,Z 138,A 136.242,B 24.9487,C -1.6541,E1 24.8771,E2 310.043} C_DIS
LIN {X -99.7272,Y 78.8523,Z 138,A 138.2784,B 24.9489,C -1.652,E1 24.8735,E2 308.0021} C_DIS
LIN {X -102.3732,Y 75.3843,Z 138,A 140.2155,B 24.9493,C -1.6452,E1 24.8703,E2 306.0718} C_DIS
LIN {X -104.7503,Y 72.0446,Z 138,A 142.0718,B 24.9496,C -1.6405,E1 24.8673,E2 304.2177} C_DIS
LIN {X -107.1956,Y 68.3535,Z 138,A 144.0749,B 24.9499,C -1.6351,E1 24.8643,E2 302.2172} C_DIS
LIN {X -109.4143,Y 64.7434,Z 138,A 146.0265,B 24.9501,C -1.6315,E1 24.8615,E2 300.2642} C_DIS
LIN {X -111.4167,Y 61.2334,Z 138,A 147.789,B 24.9506,C -1.6234,E1 24.8591,E2 298.5118} C_DIS
LIN {X -113.1648,Y 57.9342,Z 138,A 149.4136,B 24.9511,C -1.6157,E1 24.857,E2 296.8969} C_DIS
LIN {X -114.3903,Y 55.4796,Z 138,A 150.8089,B 24.9509,C -1.6192,E1 24.8553,E2 295.4856} C_DIS
LIN {X -115.9353,Y 52.1696,Z 138,A 152.2527,B 24.9517,C -1.6049,E1 24.8536,E2 294.068} C_DIS
LIN {X -117.2026,Y 49.2566,Z 138,A 153.7129,B 24.9519,C -1.6017,E1 24.852,E2 292.6073} C_DIS
LIN {X -118.3911,Y 46.3273,Z 138,A 155.2192,B 24.9519,C -1.601,E1 24.8504,E2 291.0943} C_DIS
LIN {X -119.5008,Y 43.3847,Z 138,A 156.4954,B 24.9526,C -1.5901,E1 24.8492,E2 289.8368} C_DIS
LIN {X -120.5319,Y 40.4319,Z 138,A 158.0382,B 24.9526,C -1.5917,E1 24.8478,E2 288.2814} C_DIS
LIN {X -121.3396,Y 37.9462,Z 138,A 159.3882,B 24.9523,C -1.5958,E1 24.8467,E2 286.9139} C_DIS
LIN {X -122.2921,Y 34.7495,Z 138,A 160.8258,B 24.9528,C -1.588,E1 24.8456,E2 285.4866} C_DIS
LIN {X -123.189,Y 31.4184,Z 138,A 162.2636,B 24.9534,C -1.5776,E1 24.8446,E2 284.0652} C_DIS
LIN {X -123.9127,Y 28.4304,Z 138,A 163.5916,B 24.9538,C -1.5705,E1 24.8437,E2 282.7463} C_DIS
LIN {X -124.4289,Y 26.0893,Z 138,A 164.9263,B 24.9533,C -1.5786,E1 24.8429,E2 281.3845} C_DIS
LIN {X -125.0404,Y 22.9761,Z 138,A 166.3129,B 24.9537,C -1.5719,E1 24.8422,E2 280.0055} C_DIS
LIN {X -125.5945,Y 19.7167,Z 138,A 167.5455,B 24.9547,C -1.5553,E1 24.8417,E2 278.8053} C_DIS
LIN {X -126.0201,Y 16.7832,Z 138,A 169.0917,B 24.9544,C -1.5606,E1 24.8411,E2 277.2373} C_DIS
LIN {X -126.4164,Y 13.4749,Z 138,A 170.636,B 24.9545,C -1.5576,E1 24.8406,E2 275.6909} C_DIS
LIN {X -126.7875,Y 9.3607,Z 138,A 172.427,B 24.9551,C -1.5482,E1 24.8402,E2 273.9115} C_DIS
LIN {X -126.9593,Y 6.6407,Z 138,A 173.7405,B 24.9551,C -1.5481,E1 24.8399,E2 272.5904} C_DIS
LIN {X -127.1033,Y 2.8219,Z 138,A 175.5837,B 24.9551,C -1.5479,E1 24.8399,E2 270.7364} C_DIS
LIN {X -127.1262,Y -1.4464,Z 138,A 177.4115,B 24.9557,C -1.5372,E1 24.8399,E2 268.9231} C_DIS
LIN {X -127.0452,Y -4.7206,Z 138,A 178.7596,B 24.9563,C -1.5265,E1 24.8399,E2 267.5923} C_DIS
LIN {X -126.9079,Y -7.559,Z 138,A -179.8724,B 24.9563,C -1.5264,E1 24.8401,E2 266.2166} C_DIS
LIN {X -126.681,Y -10.7049,Z 138,A -178.4007,B 24.9565,C -1.524,E1 24.8405,E2 264.7416} C_DIS
LIN {X -126.3245,Y -14.3297,Z 138,A -176.6246,B 24.9565,C -1.5249,E1 24.841,E2 262.9528} C_DIS
LIN {X -125.748,Y -18.7254,Z 138,A -174.6293,B 24.9568,C -1.5183,E1 24.8418,E2 260.9612} C_DIS
LIN {X -125.1491,Y -22.3688,Z 138,A -173.2602,B 24.9579,C -1.4995,E1 24.8424,E2 259.629} C_DIS
LIN {X -124.6335,Y -25.084,Z 138,A -171.8393,B 24.9576,C -1.5035,E1 24.8432,E2 258.1899} C_DIS
LIN {X -124.001,Y -28.0438,Z 138,A -170.4539,B 24.9578,C -1.5002,E1 24.844,E2 256.8043} C_DIS
LIN {X -123.3119,Y -30.9342,Z 138,A -169.0921,B 24.958,C -1.4971,E1 24.8449,E2 255.442} C_DIS
LIN {X -122.509,Y -33.974,Z 138,A -167.6401,B 24.9582,C -1.4943,E1 24.846,E2 253.9882} C_DIS
LIN {X -121.6233,Y -37.019,Z 138,A -166.4271,B 24.959,C -1.4799,E1 24.8469,E2 252.8025} C_DIS
LIN {X -120.8667,Y -39.4266,Z 138,A -164.9445,B 24.9583,C -1.4923,E1 24.8482,E2 251.2819} C_DIS
LIN {X -119.6863,Y -42.8701,Z 138,A -163.4416,B 24.9589,C -1.481,E1 24.8496,E2 249.7973} C_DIS
LIN {X -118.5485,Y -45.9224,Z 138,A -162.0008,B 24.9592,C -1.4754,E1 24.851,E2 248.3618} C_DIS
LIN {X -117.406,Y -48.7695,Z 138,A -160.5844,B 24.9594,C -1.4728,E1 24.8525,E2 246.9436} C_DIS
LIN {X -116.1216,Y -51.7532,Z 138,A -159.1573,B 24.9597,C -1.4669,E1 24.8541,E2 245.5229} C_DIS
LIN {X -114.8371,Y -54.5443,Z 138,A -157.7035,B 24.9597,C -1.4661,E1 24.8558,E2 244.063} C_DIS
LIN {X -113.3821,Y -57.5073,Z 138,A -156.4032,B 24.9604,C -1.4532,E1 24.8574,E2 242.7865} C_DIS
LIN {X -112.0618,Y -60.0434,Z 138,A -154.8103,B 24.9599,C -1.4637,E1 24.8595,E2 241.1601} C_DIS
LIN {X -109.9542,Y -63.8212,Z 138,A -152.8522,B 24.9601,C -1.4587,E1 24.8622,E2 239.2036} C_DIS
LIN {X -107.7265,Y -67.5145,Z 138,A -150.8637,B 24.9603,C -1.4556,E1 24.8651,E2 237.2123} C_DIS
LIN {X -105.5108,Y -70.9272,Z 138,A -149.0756,B 24.9607,C -1.4486,E1 24.8679,E2 235.4318} C_DIS
LIN {X -103.1556,Y -74.3109,Z 138,A -147.2178,B 24.9609,C -1.4439,E1 24.8709,E2 233.5762} C_DIS
LIN {X -100.7357,Y -77.5598,Z 138,A -145.3087,B 24.9609,C -1.4433,E1 24.8741,E2 231.6594} C_DIS
LIN {X -98.0776,Y -80.8942,Z 138,A -143.3827,B 24.9612,C -1.4388,E1 24.8775,E2 229.7351} C_DIS
LIN {X -95.3057,Y -84.142,Z 138,A -141.4871,B 24.9615,C -1.433,E1 24.881,E2 227.8447} C_DIS
LIN {X -92.3753,Y -87.3491,Z 138,A -139.5669,B 24.9619,C -1.4268,E1 24.8846,E2 225.9309} C_DIS
LIN {X -89.4792,Y -90.3136,Z 138,A -137.6958,B 24.9621,C -1.4229,E1 24.8883,E2 224.0611} C_DIS
LIN {X -86.7496,Y -92.9385,Z 138,A -135.9093,B 24.9621,C -1.4231,E1 24.8919,E2 222.2667} C_DIS
LIN {X -83.4967,Y -95.8715,Z 138,A -133.9538,B 24.9623,C -1.4183,E1 24.896,E2 220.315} C_DIS
LIN {X -80.2019,Y -98.6448,Z 138,A -132.004,B 24.9625,C -1.415,E1 24.9002,E2 218.3657} C_DIS
LIN {X -76.8885,Y -101.2489,Z 138,A -130.0517,B 24.9625,C -1.414,E1 24.9045,E2 216.4084} C_DIS
LIN {X -73.4742,Y -103.7528,Z 138,A -128.1385,B 24.9627,C -1.411,E1 24.9088,E2 214.4959} C_DIS
LIN {X -70.0317,Y -106.1067,Z 138,A -126.2793,B 24.9629,C -1.4069,E1 24.9131,E2 212.6402} C_DIS
LIN {X -66.3526,Y -108.4454,Z 138,A -124.3608,B 24.9632,C -1.4016,E1 24.9177,E2 210.7281} C_DIS
LIN {X -62.868,Y -110.5019,Z 138,A -122.4904,B 24.9632,C -1.4013,E1 24.9222,E2 208.8531} C_DIS
LIN {X -59.3603,Y -112.4233,Z 138,A -120.7741,B 24.9636,C -1.3947,E1 24.9264,E2 207.1476} C_DIS
LIN {X -56.9617,Y -113.6599,Z 138,A -119.3956,B 24.9632,C -1.401,E1 24.9299,E2 205.7504} C_DIS
LIN {X -53.619,Y -115.2721,Z 138,A -117.8804,B 24.9637,C -1.3913,E1 24.9337,E2 204.2543} C_DIS
LIN {X -51.0574,Y -116.4309,Z 138,A -116.5002,B 24.9635,C -1.3954,E1 24.9372,E2 202.8611} C_DIS
LIN {X -47.7745,Y -117.8145,Z 138,A -115.01,B 24.9639,C -1.3881,E1 24.941,E2 201.3849} C_DIS
LIN {X -44.8575,Y -118.9558,Z 138,A -113.5913,B 24.9639,C -1.3871,E1 24.9447,E2 199.9655} C_DIS
LIN {X -41.7749,Y -120.0728,Z 138,A -112.15,B 24.9641,C -1.384,E1 24.9485,E2 198.5287} C_DIS
LIN {X -38.8493,Y -121.0511,Z 138,A -110.77,B 24.9642,C -1.3824,E1 24.9522,E2 197.15} C_DIS
LIN {X -36.4646,Y -121.793,Z 138,A -109.4687,B 24.9638,C -1.3902,E1 24.9557,E2 195.8281} C_DIS
LIN {X -33.2781,Y -122.7008,Z 138,A -108.0109,B 24.9639,C -1.3875,E1 24.9596,E2 194.3744} C_DIS
LIN {X -29.9839,Y -123.5461,Z 138,A -106.6641,B 24.9645,C -1.3775,E1 24.9632,E2 193.0494} C_DIS
LIN {X -27.2498,Y -124.1784,Z 138,A -105.2377,B 24.9641,C -1.3848,E1 24.9671,E2 191.6039} C_DIS
LIN {X -24.1178,Y -124.824,Z 138,A -103.9534,B 24.9645,C -1.3765,E1 24.9706,E2 190.3379} C_DIS
LIN {X -21.6592,Y -125.276,Z 138,A -102.5708,B 24.9639,C -1.3887,E1 24.9745,E2 188.9249} C_DIS
LIN {X -18.5669,Y -125.7707,Z 138,A -101.2355,B 24.9641,C -1.3846,E1 24.9782,E2 187.5982} C_DIS
LIN {X -15.0856,Y -126.2343,Z 138,A -99.6999,B 24.9642,C -1.382,E1 24.9824,E2 186.0677} C_DIS
LIN {X -11.3698,Y -126.6249,Z 138,A -97.9319,B 24.964,C -1.386,E1 24.9873,E2 184.2892} C_DIS
LIN {X -8.0314,Y -126.8788,Z 138,A -96.5752,B 24.9644,C -1.3784,E1 24.9911,E2 182.9499} C_DIS
LIN {X -4.8743,Y -127.0392,Z 138,A -95.0634,B 24.9642,C -1.3829,E1 24.9953,E2 181.4271} C_DIS
LIN {X -0.7814,Y -127.1303,Z 138,A -93.2399,B 24.9642,C -1.3822,E1 25.0004,E2 179.6053} C_DIS
LIN {X -0.7814,Y -127.1303,Z 138,A -93.2399,B 24.9642,C -1.3822,E1 25.0004,E2 179.6053} C_DIS
Enddeposition()
LIN {X 0.8872,Y -126.1469,Z 138,A -92.5509,B 24.9635,C -1.3962,E1 25.0024,E2 178.883} C_DIS
Startdeposition()
$VEL.CP = VEL_PRINT
Enddeposition()
END
